C05457=1016.848,96.852,384.023,166.697,54.807,160.034
C05458=1016.842,96.602,384.039,166.694,54.816,160.035
C05459=1016.838,96.353,384.058,166.691,54.825,160.037
C05460=1016.833,96.104,384.074,166.688,54.833,160.038
C05461=1016.828,95.854,384.091,166.685,54.843,160.039
C05462=1016.822,95.605,384.108,166.683,54.852,160.040
C05463=1016.817,95.356,384.125,166.680,54.861,160.041
C05464=1016.813,95.106,384.142,166.677,54.870,160.042
C05465=1016.808,94.857,384.160,166.674,54.880,160.044
C05466=1016.802,94.608,384.177,166.671,54.888,160.045
C05467=1016.797,94.358,384.194,166.669,54.897,160.046
C05468=1016.793,94.109,384.211,166.667,54.906,160.047
C05469=1016.788,93.860,384.228,166.664,54.915,160.048
C05470=1016.783,93.610,384.245,166.661,54.925,160.050
C05471=1016.777,93.361,384.263,166.658,54.933,160.050
C05472=1016.773,93.112,384.280,166.655,54.942,160.052
C05473=1016.768,92.862,384.297,166.652,54.951,160.053
C05474=1016.763,92.613,384.314,166.650,54.961,160.054
C05475=1016.758,92.364,384.331,166.647,54.970,160.055
C05476=1016.753,92.115,384.348,166.645,54.978,160.056
C05477=1016.748,91.865,384.365,166.642,54.987,160.058
C05478=1016.743,91.615,384.382,166.639,54.997,160.059
C05479=1016.738,91.367,384.399,166.637,55.006,160.060
C05480=1016.732,91.085,384.418,166.633,55.015,160.061
C05481=1016.727,90.803,384.438,166.631,55.025,160.063
C05482=1016.722,90.522,384.457,166.627,55.036,160.064
C05483=1016.716,90.240,384.476,166.624,55.046,160.065
C05484=1016.711,89.991,384.493,166.621,55.055,160.066
C05485=1016.706,89.742,384.510,166.619,55.063,160.067
C05486=1016.701,89.492,384.527,166.616,55.073,160.069
C05487=1016.696,89.243,384.544,166.614,55.082,160.070
C05488=1016.692,88.994,384.561,166.611,55.091,160.071
C05489=1016.686,88.744,384.578,166.608,55.100,160.072
C05490=1016.681,88.494,384.594,166.605,55.109,160.073
C05491=1016.676,88.245,384.611,166.602,55.118,160.074
C05492=1016.671,87.996,384.628,166.600,55.127,160.076
C05493=1016.666,87.746,384.645,166.597,55.137,160.077
C05494=1016.661,87.497,384.661,166.594,55.146,160.078
C05495=1016.656,87.247,384.678,166.593,55.155,160.079
C05496=1016.651,86.998,384.695,166.590,55.163,160.080
C05497=1016.646,86.749,384.711,166.587,55.173,160.082
C05498=1016.640,86.500,384.728,166.584,55.182,160.083
C05499=1016.635,86.250,384.744,166.581,55.191,160.084
C05500=1016.631,86.001,384.761,166.579,55.200,160.085
C05501=1016.625,85.751,384.778,166.576,55.210,160.086
C05502=1016.620,85.502,384.795,166.573,55.218,160.087
C05503=1016.616,85.253,384.811,166.570,55.228,160.089
C05504=1016.610,85.003,384.828,166.568,55.237,160.090
C05505=1016.606,84.754,384.844,166.565,55.246,160.091
C05506=1016.601,84.504,384.861,166.562,55.255,160.092
C05507=1016.595,84.255,384.878,166.560,55.263,160.093
C05508=1016.590,84.006,384.894,166.557,55.273,160.095
C05509=1016.585,83.756,384.911,166.555,55.282,160.096
C05510=1016.580,83.507,384.927,166.552,55.291,160.097
C05511=1016.575,83.257,384.943,166.550,55.301,160.098
C05512=1016.570,83.007,384.960,166.546,55.309,160.099
C05513=1016.565,82.759,384.977,166.544,55.318,160.100
C05514=1016.560,82.509,384.994,166.541,55.328,160.102
C05515=1016.556,82.260,385.010,166.539,55.337,160.103
C05516=1016.550,82.010,385.027,166.536,55.345,160.104
C05517=1016.546,81.761,385.043,166.534,55.354,160.105
C05518=1016.540,81.512,385.060,166.531,55.364,160.106
C05519=1016.535,81.262,385.077,166.528,55.372,160.107
C05520=1016.530,81.013,385.092,166.525,55.382,160.109
C05521=1016.525,80.763,385.109,166.523,55.391,160.110
C05522=1016.521,80.514,385.126,166.521,55.400,160.111
C05523=1016.515,80.264,385.143,166.518,55.408,160.112
C05524=1016.511,80.015,385.159,166.515,55.418,160.113
C05525=1016.506,79.766,385.176,166.513,55.427,160.115
C05526=1016.501,79.516,385.192,166.509,55.436,160.116
C05527=1016.496,79.267,385.208,166.507,55.445,160.117
C05528=1016.491,79.018,385.224,166.505,55.454,160.118
C05529=1016.485,78.768,385.241,166.502,55.462,160.119
C05530=1016.481,78.519,385.258,166.499,55.472,160.120
C05531=1016.476,78.269,385.274,166.497,55.481,160.122
C05532=1016.471,78.020,385.290,166.494,55.490,160.123
C05533=1016.466,77.770,385.307,166.492,55.499,160.124
C05534=1016.461,77.521,385.324,166.489,55.507,160.125
C05535=1016.456,77.272,385.341,166.486,55.516,160.126
C05536=1016.452,77.022,385.356,166.484,55.526,160.127
C05537=1016.446,76.773,385.373,166.481,55.534,160.128
C05538=1016.441,76.524,385.389,166.478,55.544,160.130
C05539=1016.436,76.274,385.405,166.477,55.553,160.131
C05540=1016.432,76.025,385.422,166.474,55.562,160.132
C05541=1016.426,75.775,385.438,166.471,55.570,160.133
C05542=1016.422,75.526,385.454,166.468,55.580,160.134
C05543=1016.416,75.276,385.470,166.466,55.589,160.136
C05544=1016.411,74.995,385.488,166.463,55.600,160.137
C05545=1016.404,74.713,385.506,166.460,55.610,160.138
C05546=1016.399,74.432,385.525,166.457,55.619,160.139
C05547=1016.393,74.151,385.543,166.454,55.630,160.141
C05548=1016.388,73.901,385.559,166.451,55.639,160.142
C05549=1016.383,73.652,385.575,166.449,55.649,160.143
C05550=1016.378,73.402,385.591,166.445,55.657,160.144
C05551=1016.373,73.153,385.607,166.444,55.666,160.146
C05552=1016.368,72.904,385.623,166.441,55.675,160.147
C05553=1016.363,72.654,385.639,166.438,55.684,160.148
C05554=1016.358,72.405,385.655,166.436,55.693,160.149
C05555=1016.353,72.155,385.671,166.433,55.703,160.150
C05556=1016.348,71.906,385.688,166.430,55.711,160.151
C05557=1016.343,71.656,385.703,166.428,55.721,160.152
C05558=1016.338,71.407,385.720,166.426,55.730,160.154
C05559=1016.333,71.158,385.735,166.423,55.738,160.155
C05560=1016.328,70.908,385.752,166.420,55.748,160.156
C05561=1016.323,70.659,385.768,166.418,55.757,160.157
C05562=1016.318,70.409,385.784,166.415,55.766,160.158
C05563=1016.313,70.160,385.800,166.412,55.775,160.159
C05564=1016.308,69.911,385.815,166.411,55.784,160.161
C05565=1016.303,69.661,385.832,166.408,55.793,160.162
C05566=1016.298,69.412,385.847,166.405,55.802,160.163
C05567=1016.293,69.162,385.864,166.403,55.811,160.164
C05568=1016.288,68.912,385.880,166.399,55.820,160.165
C05569=1016.283,68.664,385.896,166.397,55.829,160.167
C05570=1016.278,68.414,385.912,166.395,55.837,160.168
C05571=1016.273,68.164,385.927,166.392,55.847,160.169
C05572=1016.269,67.915,385.943,166.390,55.856,160.170
C05573=1016.263,67.665,385.959,166.387,55.865,160.171
C05574=1016.259,67.416,385.975,166.384,55.874,160.172
C05575=1016.253,67.167,385.991,166.382,55.884,160.174
C05576=1016.248,66.917,386.006,166.380,55.892,160.175
C05577=1016.243,66.668,386.022,166.377,55.901,160.176
C05578=1016.237,66.418,386.038,166.375,55.911,160.177
C05579=1016.233,66.169,386.054,166.372,55.919,160.178
C05580=1016.228,65.919,386.069,166.369,55.929,160.179
C05581=1016.222,65.670,386.085,166.367,55.938,160.181
C05582=1016.218,65.420,386.101,166.364,55.947,160.182
C05583=1016.213,65.171,386.116,166.362,55.956,160.183
C05584=1016.208,64.921,386.132,166.359,55.964,160.184
C05585=1016.202,64.672,386.148,166.357,55.974,160.185
C05586=1016.197,64.423,386.163,166.354,55.983,160.187
C05587=1016.192,64.173,386.180,166.351,55.992,160.188
C05588=1016.187,63.923,386.195,166.349,56.001,160.189
C05589=1016.182,63.674,386.210,166.346,56.011,160.190
C05590=1016.178,63.425,386.226,166.344,56.019,160.191
C05591=1016.172,63.175,386.242,166.342,56.028,160.192
C05592=1016.167,62.926,386.257,166.339,56.037,160.193
C05593=1016.163,62.676,386.273,166.336,56.046,160.195
C05594=1016.157,62.426,386.288,166.334,56.056,160.196
C05595=1016.152,62.177,386.304,166.331,56.064,160.197
C05596=1016.147,61.928,386.319,166.328,56.074,160.198
C05597=1016.141,61.678,386.334,166.326,56.083,160.199
C05598=1016.136,61.429,386.349,166.323,56.093,160.201
C05599=1016.131,61.179,386.365,166.320,56.101,160.202
C05600=1016.126,60.930,386.380,166.318,56.111,160.203
C05601=1016.121,60.680,386.395,166.316,56.120,160.204
C05602=1016.116,60.431,386.411,166.314,56.129,160.206
C05603=1016.111,60.182,386.426,166.311,56.138,160.206
C05604=1016.105,59.932,386.441,166.308,56.147,160.208
C05605=1016.100,59.682,386.456,166.306,56.157,160.209
C05606=1016.096,59.433,386.472,166.303,56.166,160.210
C05607=1016.090,59.184,386.487,166.300,56.175,160.211
C05608=1016.084,58.903,386.504,166.298,56.185,160.213
C05609=1016.079,58.621,386.521,166.295,56.196,160.214
C05610=1016.073,58.340,386.539,166.293,56.206,160.215
C05611=1016.067,58.058,386.556,166.289,56.216,160.217
C05612=1016.062,57.808,386.571,166.287,56.225,160.218
C05613=1016.057,57.559,386.587,166.284,56.235,160.219
C05614=1016.052,57.310,386.602,166.281,56.243,160.220
C05615=1016.047,57.060,386.617,166.279,56.253,160.221
C05616=1016.042,56.811,386.632,166.276,56.262,160.223
C05617=1016.036,56.561,386.648,166.273,56.271,160.224
C05618=1016.031,56.312,386.663,166.272,56.280,160.225
C05619=1016.026,56.063,386.678,166.269,56.289,160.226
C05620=1016.021,55.813,386.693,166.267,56.298,160.227
C05621=1016.016,55.563,386.708,166.264,56.307,160.228
C05622=1016.010,55.314,386.723,166.261,56.316,160.229
C05623=1016.005,55.064,386.738,166.259,56.326,160.231
C05624=1016.000,54.815,386.754,166.256,56.334,160.232
C05625=1015.995,54.566,386.769,166.253,56.344,160.233
C05626=1015.990,54.316,386.784,166.252,56.352,160.234
C05627=1015.985,54.067,386.799,166.249,56.361,160.235
C05628=1015.980,53.817,386.814,166.246,56.370,160.236
C05629=1015.975,53.567,386.829,166.244,56.380,160.238
C05630=1015.970,53.318,386.844,166.241,56.388,160.239
C05631=1015.965,53.069,386.859,166.238,56.398,160.240
C05632=1015.960,52.820,386.875,166.237,56.406,160.241
C05633=1015.955,52.570,386.890,166.234,56.416,160.242
C05634=1015.950,52.320,386.904,166.231,56.424,160.243
C05635=1015.945,52.070,386.920,166.229,56.434,160.245
C05636=1015.940,51.821,386.936,166.226,56.442,160.246
C05637=1015.935,51.572,386.951,166.225,56.452,160.247
C05638=1015.930,51.322,386.966,166.222,56.460,160.248
C05639=1015.925,51.072,386.980,166.219,56.470,160.249
C05640=1015.920,50.823,386.996,166.216,56.478,160.250
C05641=1015.915,50.574,387.011,166.214,56.488,160.252
C05642=1015.910,50.325,387.026,166.212,56.496,160.253
C05643=1015.905,50.074,387.041,166.209,56.505,160.254
C05644=1015.900,49.825,387.056,166.207,56.514,160.255
C05645=1015.895,49.575,387.071,166.204,56.523,160.256
C05646=1015.889,49.326,387.086,166.201,56.533,160.257
C05647=1015.885,49.076,387.101,166.200,56.541,160.258
C05648=1015.880,48.827,387.116,166.197,56.550,160.259
C05649=1015.875,48.578,387.131,166.194,56.559,160.261
C05650=1015.870,48.329,387.146,166.191,56.568,160.262
C05651=1015.865,48.079,387.161,166.189,56.576,160.263
C05652=1015.860,47.829,387.176,166.187,56.586,160.264
C05653=1015.855,47.580,387.191,166.184,56.594,160.265
C05654=1015.850,47.331,387.206,166.181,56.603,160.266
C05655=1015.845,47.081,387.221,166.180,56.612,160.268
C05656=1015.839,46.831,387.236,166.177,56.621,160.268
C05657=1015.834,46.582,387.251,166.174,56.630,160.269
C05658=1015.830,46.332,387.266,166.171,56.639,160.270
C05659=1015.825,46.083,387.281,166.170,56.648,160.272
C05660=1015.819,45.833,387.296,166.167,56.656,160.273
C05661=1015.815,45.583,387.311,166.164,56.665,160.274
C05662=1015.810,45.334,387.326,166.163,56.674,160.275
C05663=1015.805,45.085,387.341,166.160,56.683,160.276
C05664=1015.800,44.835,387.355,166.157,56.692,160.277
C05665=1015.795,44.586,387.371,166.154,56.701,160.278
C05666=1015.790,44.336,387.386,166.152,56.709,160.280
C05667=1015.785,44.087,387.400,166.150,56.718,160.281
C05668=1015.780,43.837,387.415,166.147,56.727,160.282
C05669=1015.775,43.587,387.430,166.145,56.736,160.283
C05670=1015.770,43.338,387.445,166.143,56.744,160.284
C05671=1015.765,43.089,387.460,166.140,56.753,160.285
C05672=1015.760,42.831,387.476,166.138,56.762,160.286
C05673=1015.755,42.574,387.491,166.135,56.771,160.287
C05674=1015.751,42.315,387.506,166.133,56.780,160.289
C05675=1015.745,42.058,387.521,166.130,56.789,160.290
C05676=1015.740,41.809,387.536,166.127,56.798,160.291
C05677=1015.735,41.559,387.551,166.125,56.807,160.292
C05678=1015.730,41.310,387.565,166.122,56.816,160.293
C05679=1015.725,41.060,387.580,166.120,56.825,160.294
C05680=1015.720,40.810,387.594,166.118,56.834,160.295
C05681=1015.715,40.561,387.610,166.115,56.843,160.296
C05682=1015.710,40.311,387.623,166.112,56.852,160.297
C05683=1015.705,40.062,387.639,166.111,56.861,160.299
C05684=1015.701,39.813,387.653,166.108,56.870,160.300
C05685=1015.695,39.563,387.667,166.105,56.878,160.301
C05686=1015.690,39.314,387.682,166.103,56.887,160.302
C05687=1015.685,39.064,387.696,166.101,56.896,160.303
C05688=1015.680,38.815,387.711,166.099,56.905,160.304
C05689=1015.675,38.565,387.725,166.096,56.914,160.305
C05690=1015.670,38.315,387.740,166.093,56.923,160.306
C05691=1015.665,38.066,387.755,166.092,56.932,160.308
C05692=1015.660,37.816,387.769,166.089,56.941,160.309
C05693=1015.655,37.567,387.783,166.086,56.949,160.310
C05694=1015.650,37.317,387.798,166.083,56.958,160.311
C05695=1015.645,37.068,387.813,166.081,56.967,160.312
C05696=1015.639,36.818,387.827,166.079,56.976,160.313
C05697=1015.635,36.568,387.841,166.076,56.985,160.314
C05698=1015.630,36.319,387.856,166.074,56.993,160.316
C05699=1015.625,36.070,387.870,166.072,57.002,160.317
C05700=1015.620,35.820,387.884,166.069,57.012,160.318
C05701=1015.615,35.571,387.898,166.067,57.020,160.319
C05702=1015.610,35.321,387.913,166.064,57.029,160.320
C05703=1015.604,35.072,387.927,166.061,57.038,160.321
C05704=1015.599,34.822,387.942,166.060,57.047,160.322
C05705=1015.594,34.572,387.956,166.057,57.056,160.323
C05706=1015.589,34.322,387.970,166.054,57.065,160.324
C05707=1015.584,34.073,387.983,166.051,57.074,160.325
C05708=1015.580,33.824,387.998,166.049,57.083,160.327
C05709=1015.574,33.574,388.012,166.047,57.092,160.328
C05710=1015.569,33.325,388.027,166.044,57.100,160.329
C05711=1015.564,33.075,388.041,166.042,57.109,160.330
C05712=1015.558,32.826,388.055,166.039,57.119,160.331
C05713=1015.553,32.576,388.069,166.038,57.127,160.332
C05714=1015.548,32.327,388.083,166.035,57.136,160.333
C05715=1015.544,32.077,388.097,166.032,57.145,160.334
C05716=1015.538,31.827,388.111,166.029,57.154,160.335
C05717=1015.533,31.577,388.125,166.028,57.163,160.337
C05718=1015.528,31.328,388.139,166.025,57.172,160.338
C05719=1015.523,31.078,388.154,166.023,57.181,160.339
C05720=1015.518,30.829,388.167,166.020,57.189,160.340
C05721=1015.513,30.580,388.182,166.018,57.198,160.341
C05722=1015.508,30.330,388.196,166.015,57.207,160.342
C05723=1015.503,30.080,388.211,166.012,57.215,160.343
C05724=1015.498,29.807,388.226,166.010,57.225,160.345
C05725=1015.492,29.534,388.241,166.007,57.235,160.346
C05726=1015.487,29.260,388.256,166.005,57.245,160.347
C05727=1015.481,28.987,388.271,166.003,57.254,160.348
C05728=1015.476,28.737,388.286,166.000,57.263,160.349
C05729=1015.471,28.488,388.299,165.997,57.272,160.350
C05730=1015.467,28.238,388.314,165.995,57.280,160.352
C05731=1015.461,27.989,388.328,165.993,57.289,160.353
C05732=1015.456,27.739,388.342,165.990,57.298,160.354
C05733=1015.451,27.490,388.356,165.988,57.306,160.355
C05734=1015.446,27.240,388.370,165.985,57.315,160.356
C05735=1015.441,26.990,388.384,165.983,57.324,160.357
C05736=1015.436,26.710,388.400,165.980,57.334,160.358
C05737=1015.429,26.428,388.415,165.977,57.344,160.359
C05738=1015.423,26.147,388.431,165.975,57.355,160.361
C05739=1015.418,25.866,388.446,165.972,57.364,160.362
C05740=1015.413,25.616,388.460,165.970,57.373,160.363
C05741=1015.408,25.366,388.475,165.967,57.382,160.364
C05742=1015.403,25.116,388.488,165.965,57.390,160.365
C05743=1015.398,24.867,388.501,165.962,57.399,160.366
C05744=1015.392,24.618,388.515,165.960,57.408,160.367
C05745=1015.388,24.368,388.530,165.957,57.417,160.368
C05746=1015.383,24.119,388.543,165.955,57.425,160.369
C05747=1015.378,23.869,388.556,165.953,57.434,160.370
C05748=1015.372,23.619,388.570,165.950,57.443,160.371
C05749=1015.367,23.370,388.584,165.947,57.452,160.373
C05750=1015.363,23.120,388.598,165.945,57.460,160.374
C05751=1015.357,22.871,388.612,165.943,57.469,160.375
C05752=1015.352,22.621,388.625,165.940,57.478,160.376
C05753=1015.347,22.372,388.639,165.938,57.487,160.377
C05754=1015.342,22.122,388.652,165.935,57.495,160.378
C05755=1015.337,21.872,388.666,165.933,57.504,160.379
C05756=1015.332,21.623,388.680,165.930,57.513,160.380
C05757=1015.327,21.373,388.693,165.928,57.522,160.381
C05758=1015.321,21.124,388.707,165.926,57.531,160.382
C05759=1015.317,20.874,388.720,165.923,57.539,160.383
C05760=1015.312,20.624,388.735,165.921,57.548,160.385
C05761=1015.307,20.375,388.748,165.919,57.557,160.386
C05762=1015.302,20.125,388.761,165.916,57.566,160.387
C05763=1015.297,19.876,388.775,165.914,57.574,160.388
C05764=1015.291,19.626,388.789,165.912,57.583,160.389
C05765=1015.287,19.377,388.803,165.908,57.591,160.390
C05766=1015.282,19.127,388.816,165.907,57.600,160.391
C05767=1015.277,18.878,388.830,165.904,57.609,160.392
C05768=1015.272,18.628,388.843,165.901,57.617,160.393
C05769=1015.266,18.378,388.857,165.900,57.626,160.394
C05770=1015.261,18.129,388.870,165.897,57.635,160.395
C05771=1015.256,17.879,388.883,165.894,57.644,160.396
C05772=1015.251,17.630,388.897,165.893,57.652,160.397
C05773=1015.246,17.380,388.910,165.890,57.661,160.398
C05774=1015.241,17.130,388.924,165.887,57.670,160.399
C05775=1015.236,16.881,388.937,165.884,57.679,160.400
C05776=1015.231,16.631,388.951,165.882,57.687,160.401
C05777=1015.227,16.381,388.964,165.880,57.696,160.402
C05778=1015.221,16.132,388.978,165.877,57.704,160.403
C05779=1015.216,15.882,388.992,165.875,57.713,160.405
C05780=1015.211,15.633,389.004,165.873,57.722,160.406
C05781=1015.206,15.383,389.018,165.870,57.731,160.407
C05782=1015.201,15.134,389.031,165.868,57.739,160.408
C05783=1015.196,14.884,389.045,165.865,57.747,160.409
C05784=1015.191,14.635,389.058,165.863,57.756,160.410
C05785=1015.186,14.385,389.072,165.861,57.765,160.411
C05786=1015.181,14.135,389.085,165.858,57.774,160.412
C05787=1015.176,13.886,389.098,165.856,57.781,160.413
C05788=1015.170,13.636,389.111,165.853,57.790,160.414
C05789=1015.166,13.386,389.124,165.850,57.799,160.415
C05790=1015.160,13.137,389.138,165.849,57.808,160.416
C05791=1015.156,12.887,389.151,165.846,57.817,160.417
C05792=1015.151,12.637,389.164,165.844,57.826,160.418
C05793=1015.145,12.388,389.178,165.841,57.833,160.419
C05794=1015.140,12.138,389.190,165.839,57.842,160.420
C05795=1015.135,11.888,389.203,165.836,57.851,160.421
C05796=1015.130,11.639,389.217,165.833,57.860,160.422
C05797=1015.125,11.389,389.230,165.832,57.869,160.424
C05798=1015.119,11.140,389.242,165.829,57.878,160.425
C05799=1015.114,10.890,389.255,165.827,57.887,160.426
C05800=1015.108,10.610,389.270,165.825,57.896,160.427
C05801=1015.103,10.331,389.285,165.821,57.906,160.428
C05802=1015.097,10.051,389.298,165.819,57.915,160.429
C05803=1015.091,9.771,389.313,165.816,57.925,160.430
C05804=1015.086,9.521,389.327,165.813,57.934,160.431
C05805=1015.082,9.272,389.339,165.811,57.942,160.432
C05806=1015.076,9.022,389.353,165.808,57.951,160.433
C05807=1015.071,8.773,389.365,165.806,57.960,160.434
C05808=1015.066,8.523,389.379,165.804,57.968,160.436
C05809=1015.061,8.273,389.391,165.801,57.977,160.436
C05810=1015.056,8.024,389.404,165.798,57.986,160.437
C05811=1015.050,7.774,389.417,165.797,57.994,160.439
C05812=1015.046,7.525,389.430,165.794,58.003,160.440
C05813=1015.041,7.275,389.443,165.791,58.011,160.440
C05814=1015.035,7.026,389.456,165.789,58.020,160.442
C05815=1015.030,6.775,389.469,165.787,58.029,160.443
C05816=1015.026,6.526,389.481,165.784,58.037,160.444
C05817=1015.021,6.276,389.494,165.782,58.046,160.445
C05818=1015.015,6.027,389.508,165.779,58.054,160.446
C05819=1015.010,5.778,389.520,165.777,58.062,160.447
C05820=1015.005,5.527,389.533,165.774,58.071,160.448
C05821=1015.001,5.278,389.546,165.773,58.080,160.449
C05822=1014.995,5.028,389.559,165.770,58.088,160.450
C05823=1014.990,4.779,389.572,165.767,58.097,160.451
C05824=1014.986,4.529,389.584,165.765,58.105,160.452
C05825=1014.980,4.279,389.598,165.762,58.114,160.453
C05826=1014.975,4.030,389.610,165.761,58.122,160.454
C05827=1014.970,3.781,389.623,165.758,58.130,160.455
C05828=1014.965,3.531,389.636,165.755,58.139,160.456
C05829=1014.960,3.281,389.649,165.753,58.147,160.457
C05830=1014.955,3.031,389.662,165.750,58.156,160.458
C05831=1014.950,2.782,389.674,165.748,58.164,160.459
C05832=1014.945,2.532,389.687,165.746,58.173,160.460
C05833=1014.940,2.282,389.700,165.743,58.181,160.461
C05834=1014.935,2.033,389.713,165.741,58.190,160.462
C05835=1014.930,1.783,389.725,165.739,58.198,160.463
C05836=1014.925,1.533,389.739,165.736,58.206,160.464
C05837=1014.920,1.284,389.751,165.734,58.214,160.465
C05838=1014.915,1.035,389.763,165.731,58.223,160.465
C05839=1014.910,0.784,389.777,165.729,58.231,160.467
C05840=1014.906,0.535,389.789,165.726,58.239,160.467
C05841=1014.900,0.286,389.802,165.725,58.248,160.469
C05842=1014.895,0.035,389.815,165.722,58.256,160.469
C05843=1014.890,-0.214,389.828,165.719,58.264,160.470
C05844=1014.886,-0.464,389.840,165.717,58.273,160.471
C05845=1014.880,-0.713,389.853,165.715,58.281,160.472
C05846=1014.875,-0.963,389.866,165.712,58.290,160.473
C05847=1014.871,-1.212,389.878,165.710,58.298,160.474
C05848=1014.866,-1.462,389.891,165.707,58.306,160.475
C05849=1014.860,-1.712,389.904,165.705,58.314,160.476
C05850=1014.856,-1.961,389.917,165.702,58.323,160.477
C05851=1014.851,-2.211,389.929,165.700,58.330,160.478
C05852=1014.845,-2.461,389.942,165.697,58.339,160.479
C05853=1014.841,-2.710,389.955,165.695,58.347,160.480
C05854=1014.836,-2.960,389.967,165.693,58.355,160.481
C05855=1014.832,-3.209,389.980,165.690,58.363,160.482
C05856=1014.826,-3.459,389.993,165.688,58.371,160.483
C05857=1014.821,-3.708,390.006,165.686,58.380,160.484
C05858=1014.817,-3.958,390.018,165.683,58.388,160.485
C05859=1014.812,-4.207,390.031,165.680,58.396,160.485
C05860=1014.806,-4.458,390.043,165.678,58.404,160.486
C05861=1014.802,-4.707,390.056,165.677,58.413,160.487
C05862=1014.797,-4.957,390.068,165.674,58.421,160.488
C05863=1014.792,-5.206,390.081,165.670,58.429,160.489
C05864=1014.786,-5.484,390.094,165.669,58.439,160.490
C05865=1014.781,-5.762,390.107,165.666,58.448,160.491
C05866=1014.775,-6.039,390.121,165.663,58.457,160.492
C05867=1014.769,-6.317,390.135,165.660,58.466,160.493
C05868=1014.764,-6.566,390.146,165.658,58.475,160.495
C05869=1014.759,-6.817,390.160,165.655,58.483,160.495
C05870=1014.754,-7.066,390.172,165.653,58.491,160.496
C05871=1014.749,-7.316,390.183,165.651,58.500,160.497
C05872=1014.744,-7.565,390.196,165.649,58.508,160.498
C05873=1014.739,-7.815,390.207,165.646,58.516,160.499
C05874=1014.733,-8.065,390.220,165.644,58.525,160.500
C05875=1014.729,-8.314,390.233,165.641,58.533,160.501
C05876=1014.724,-8.564,390.244,165.639,58.541,160.502
C05877=1014.718,-8.813,390.256,165.636,58.549,160.503
C05878=1014.714,-9.063,390.269,165.634,58.558,160.504
C05879=1014.709,-9.313,390.281,165.631,58.566,160.505
C05880=1014.704,-9.563,390.294,165.629,58.574,160.506
C05881=1014.699,-9.813,390.305,165.626,58.582,160.506
C05882=1014.693,-10.062,390.318,165.625,58.591,160.508
C05883=1014.689,-10.312,390.330,165.621,58.599,160.508
C05884=1014.684,-10.561,390.342,165.619,58.607,160.509
C05885=1014.678,-10.810,390.354,165.616,58.615,160.510
C05886=1014.674,-11.060,390.366,165.614,58.623,160.511
C05887=1014.668,-11.310,390.379,165.612,58.631,160.512
C05888=1014.663,-11.560,390.390,165.610,58.640,160.513
C05889=1014.659,-11.810,390.403,165.608,58.648,160.514
C05890=1014.654,-12.059,390.414,165.605,58.656,160.515
C05891=1014.648,-12.309,390.427,165.602,58.664,160.516
C05892=1014.644,-12.559,390.439,165.600,58.672,160.517
C05893=1014.639,-12.808,390.451,165.597,58.680,160.518
C05894=1014.634,-13.058,390.462,165.595,58.688,160.518
C05895=1014.629,-13.307,390.475,165.592,58.696,160.519
C05896=1014.624,-13.557,390.487,165.590,58.704,160.520
C05897=1014.619,-13.806,390.499,165.588,58.712,160.521
C05898=1014.614,-14.057,390.511,165.585,58.720,160.522
C05899=1014.609,-14.306,390.523,165.583,58.728,160.523
C05900=1014.604,-14.556,390.535,165.581,58.736,160.524
C05901=1014.599,-14.805,390.548,165.578,58.744,160.525
C05902=1014.594,-15.055,390.559,165.576,58.752,160.526
C05903=1014.589,-15.305,390.571,165.574,58.760,160.526
C05904=1014.585,-15.554,390.583,165.571,58.768,160.527
C05905=1014.580,-15.804,390.595,165.569,58.776,160.528
C05906=1014.575,-16.054,390.608,165.567,58.784,160.529
C05907=1014.570,-16.304,390.619,165.564,58.792,160.530
C05908=1014.565,-16.553,390.630,165.562,58.800,160.531
C05909=1014.560,-16.803,390.642,165.559,58.809,160.532
C05910=1014.555,-17.052,390.654,165.557,58.817,160.533
C05911=1014.550,-17.302,390.666,165.553,58.825,160.533
C05912=1014.545,-17.552,390.677,165.551,58.833,160.534
C05913=1014.540,-17.802,390.689,165.549,58.841,160.535
C05914=1014.534,-18.051,390.701,165.546,58.849,160.536
C05915=1014.529,-18.301,390.712,165.544,58.857,160.537
C05916=1014.524,-18.551,390.724,165.541,58.865,160.538
C05917=1014.519,-18.800,390.735,165.539,58.873,160.539
C05918=1014.515,-19.050,390.748,165.537,58.881,160.540
C05919=1014.510,-19.300,390.759,165.534,58.889,160.540
C05920=1014.505,-19.549,390.771,165.532,58.897,160.541
C05921=1014.500,-19.799,390.782,165.530,58.905,160.542
C05922=1014.495,-20.049,390.794,165.527,58.913,160.543
C05923=1014.489,-20.298,390.806,165.525,58.921,160.544
C05924=1014.484,-20.548,390.818,165.523,58.929,160.545
C05925=1014.479,-20.798,390.829,165.520,58.937,160.546
C05926=1014.474,-21.048,390.840,165.518,58.945,160.547
C05927=1014.469,-21.297,390.852,165.516,58.953,160.548
C05928=1014.464,-21.573,390.865,165.513,58.962,160.548
C05929=1014.458,-21.849,390.878,165.511,58.971,160.550
C05930=1014.453,-22.125,390.891,165.508,58.979,160.550
C05931=1014.448,-22.401,390.903,165.505,58.988,160.551
C05932=1014.443,-22.651,390.915,165.502,58.996,160.552
C05933=1014.438,-22.900,390.927,165.499,59.004,160.553
C05934=1014.433,-23.150,390.938,165.498,59.011,160.554
C05935=1014.428,-23.399,390.950,165.496,59.019,160.555
C05936=1014.423,-23.649,390.961,165.492,59.028,160.555
C05937=1014.418,-23.899,390.973,165.490,59.035,160.556
C05938=1014.413,-24.148,390.984,165.488,59.043,160.557
C05939=1014.408,-24.398,390.995,165.486,59.051,160.558
C05940=1014.403,-24.648,391.007,165.483,59.059,160.559
C05941=1014.398,-24.897,391.018,165.480,59.066,160.559
C05942=1014.393,-25.147,391.030,165.478,59.074,160.560
C05943=1014.388,-25.397,391.041,165.476,59.082,160.561
C05944=1014.383,-25.647,391.053,165.473,59.090,160.562
C05945=1014.378,-25.897,391.064,165.471,59.097,160.563
C05946=1014.374,-26.146,391.075,165.469,59.105,160.564
C05947=1014.369,-26.395,391.088,165.466,59.113,160.564
C05948=1014.364,-26.645,391.100,165.464,59.120,160.565
C05949=1014.359,-26.895,391.111,165.462,59.128,160.566
C05950=1014.354,-27.145,391.122,165.459,59.136,160.567
C05951=1014.349,-27.394,391.134,165.456,59.143,160.567
C05952=1014.345,-27.644,391.145,165.454,59.151,160.568
C05953=1014.340,-27.894,391.156,165.452,59.159,160.569
C05954=1014.335,-28.144,391.167,165.449,59.166,160.570
C05955=1014.329,-28.393,391.178,165.446,59.175,160.571
C05956=1014.324,-28.643,391.190,165.445,59.182,160.572
C05957=1014.319,-28.893,391.201,165.442,59.190,160.572
C05958=1014.315,-29.142,391.212,165.440,59.198,160.573
C05959=1014.310,-29.392,391.222,165.437,59.206,160.574
C05960=1014.305,-29.642,391.234,165.434,59.213,160.575
C05961=1014.300,-29.892,391.245,165.432,59.221,160.576
C05962=1014.295,-30.141,391.257,165.431,59.229,160.577
C05963=1014.290,-30.391,391.268,165.427,59.237,160.577
C05964=1014.285,-30.641,391.278,165.425,59.244,160.578
C05965=1014.280,-30.890,391.290,165.422,59.252,160.579
C05966=1014.275,-31.140,391.301,165.420,59.260,160.580
C05967=1014.270,-31.389,391.312,165.417,59.268,160.580
C05968=1014.265,-31.640,391.322,165.415,59.275,160.581
C05969=1014.260,-31.889,391.334,165.413,59.283,160.582
C05970=1014.255,-32.139,391.345,165.410,59.290,160.583
C05971=1014.251,-32.388,391.356,165.408,59.298,160.584
C05972=1014.245,-32.638,391.366,165.406,59.305,160.584
C05973=1014.240,-32.888,391.378,165.403,59.314,160.585
C05974=1014.236,-33.137,391.389,165.400,59.321,160.586
C05975=1014.231,-33.388,391.400,165.398,59.329,160.587
C05976=1014.225,-33.637,391.411,165.396,59.336,160.587
C05977=1014.220,-33.887,391.422,165.393,59.343,160.588
C05978=1014.216,-34.136,391.433,165.391,59.351,160.589
C05979=1014.211,-34.386,391.444,165.389,59.358,160.590
C05980=1014.205,-34.636,391.455,165.387,59.366,160.591
C05981=1014.201,-34.885,391.466,165.383,59.374,160.591
C05982=1014.196,-35.135,391.477,165.381,59.381,160.592
C05983=1014.191,-35.385,391.488,165.379,59.389,160.593
C05984=1014.186,-35.634,391.499,165.376,59.396,160.593
C05985=1014.182,-35.884,391.510,165.374,59.404,160.594
C05986=1014.177,-36.134,391.521,165.372,59.411,160.595
C05987=1014.172,-36.384,391.531,165.369,59.419,160.596
C05988=1014.167,-36.633,391.542,165.367,59.426,160.596
C05989=1014.162,-36.883,391.554,165.365,59.434,160.597
C05990=1014.158,-37.133,391.564,165.362,59.441,160.598
C05991=1014.153,-37.383,391.576,165.360,59.448,160.599
C05992=1014.147,-37.657,391.588,165.357,59.457,160.599
C05993=1014.142,-37.932,391.600,165.355,59.465,160.600
C05994=1014.137,-38.208,391.612,165.352,59.473,160.601
C05995=1014.131,-38.482,391.623,165.348,59.481,160.601
C05996=1014.126,-38.731,391.634,165.347,59.488,160.603
C05997=1014.121,-38.982,391.645,165.345,59.495,160.603
C05998=1014.116,-39.231,391.656,165.342,59.503,160.604
C05999=1014.112,-39.481,391.666,165.340,59.510,160.605
C06000=1014.107,-39.731,391.678,165.337,59.517,160.605
C06001=1014.103,-39.980,391.688,165.334,59.525,160.606
C06002=1014.097,-40.230,391.699,165.332,59.533,160.607
C06003=1014.091,-40.480,391.709,165.329,59.540,160.607
C06004=1014.087,-40.730,391.719,165.327,59.547,160.608
C06005=1014.081,-40.979,391.730,165.325,59.555,160.609
C06006=1014.077,-41.229,391.741,165.322,59.562,160.610
C06007=1014.072,-41.479,391.751,165.320,59.569,160.610
C06008=1014.068,-41.728,391.762,165.317,59.577,160.611
C06009=1014.062,-41.978,391.772,165.315,59.585,160.612
C06010=1014.058,-42.227,391.783,165.313,59.592,160.613
C06011=1014.052,-42.477,391.793,165.310,59.599,160.613
C06012=1014.048,-42.728,391.804,165.308,59.606,160.614
C06013=1014.042,-42.977,391.815,165.305,59.613,160.615
C06014=1014.038,-43.227,391.825,165.303,59.621,160.615
C06015=1014.033,-43.476,391.835,165.300,59.628,160.616
C06016=1014.028,-43.727,391.846,165.298,59.636,160.617
C06017=1014.023,-43.976,391.857,165.296,59.643,160.618
C06018=1014.018,-44.226,391.867,165.293,59.650,160.618
C06019=1014.014,-44.475,391.877,165.291,59.658,160.619
C06020=1014.008,-44.725,391.888,165.288,59.665,160.619
C06021=1014.004,-44.975,391.898,165.286,59.672,160.620
C06022=1013.998,-45.225,391.909,165.283,59.679,160.621
C06023=1013.994,-45.474,391.919,165.282,59.686,160.622
C06024=1013.988,-45.724,391.930,165.279,59.693,160.622
C06025=1013.984,-45.974,391.940,165.277,59.700,160.623
C06026=1013.979,-46.224,391.950,165.274,59.708,160.624
C06027=1013.975,-46.473,391.961,165.272,59.715,160.624
C06028=1013.970,-46.722,391.971,165.269,59.722,160.625
C06029=1013.965,-46.973,391.982,165.267,59.729,160.626
C06030=1013.960,-47.222,391.992,165.263,59.736,160.626
C06031=1013.956,-47.473,392.003,165.262,59.743,160.627
C06032=1013.951,-47.722,392.012,165.259,59.750,160.627
C06033=1013.945,-47.971,392.023,165.257,59.757,160.628
C06034=1013.941,-48.221,392.034,165.254,59.764,160.629
C06035=1013.935,-48.471,392.044,165.252,59.772,160.629
C06036=1013.931,-48.721,392.054,165.249,59.779,160.630
C06037=1013.926,-48.970,392.064,165.247,59.785,160.631
C06038=1013.921,-49.220,392.075,165.245,59.792,160.631
C06039=1013.917,-49.470,392.085,165.242,59.799,160.632
C06040=1013.912,-49.720,392.096,165.240,59.807,160.633
C06041=1013.907,-49.969,392.106,165.237,59.814,160.633
C06042=1013.903,-50.219,392.116,165.235,59.820,160.634
C06043=1013.898,-50.469,392.126,165.233,59.827,160.634
C06044=1013.893,-50.719,392.137,165.230,59.834,160.635
C06045=1013.888,-50.969,392.147,165.227,59.841,160.635
C06046=1013.884,-51.219,392.157,165.226,59.848,160.636
C06047=1013.879,-51.469,392.167,165.223,59.855,160.637
C06048=1013.874,-51.718,392.177,165.221,59.862,160.638
C06049=1013.869,-51.968,392.187,165.218,59.869,160.638
C06050=1013.863,-52.218,392.197,165.216,59.877,160.639
C06051=1013.859,-52.467,392.207,165.213,59.884,160.639
C06052=1013.854,-52.717,392.217,165.211,59.891,160.640
C06053=1013.849,-52.967,392.226,165.208,59.898,160.640
C06054=1013.844,-53.217,392.236,165.206,59.904,160.641
C06055=1013.839,-53.466,392.246,165.204,59.912,160.642
C06056=1013.833,-53.741,392.257,165.201,59.920,160.643
C06057=1013.828,-54.016,392.268,165.198,59.927,160.643
C06058=1013.823,-54.291,392.279,165.195,59.935,160.644
C06059=1013.817,-54.567,392.289,165.193,59.943,160.645
C06060=1013.812,-54.817,392.299,165.190,59.950,160.645
C06061=1013.807,-55.066,392.309,165.187,59.957,160.646
C06062=1013.802,-55.315,392.319,165.186,59.964,160.647
C06063=1013.797,-55.565,392.328,165.183,59.971,160.647
C06064=1013.792,-55.816,392.338,165.180,59.978,160.648
C06065=1013.787,-56.065,392.348,165.178,59.985,160.648
C06066=1013.783,-56.314,392.357,165.175,59.992,160.649
C06067=1013.777,-56.565,392.368,165.173,59.998,160.649
C06068=1013.773,-56.815,392.377,165.171,60.005,160.650
C06069=1013.768,-57.064,392.386,165.168,60.013,160.651
C06070=1013.764,-57.314,392.397,165.166,60.019,160.651
C06071=1013.758,-57.564,392.407,165.164,60.026,160.652
C06072=1013.754,-57.814,392.416,165.161,60.033,160.653
C06073=1013.749,-58.063,392.426,165.158,60.040,160.653
C06074=1013.744,-58.313,392.436,165.157,60.047,160.654
C06075=1013.740,-58.563,392.445,165.154,60.053,160.654
C06076=1013.734,-58.813,392.455,165.151,60.060,160.655
C06077=1013.729,-59.062,392.465,165.149,60.066,160.655
C06078=1013.724,-59.312,392.475,165.147,60.074,160.656
C06079=1013.720,-59.562,392.484,165.144,60.080,160.656
C06080=1013.714,-59.812,392.494,165.142,60.087,160.657
C06081=1013.710,-60.061,392.504,165.139,60.094,160.658
C06082=1013.705,-60.311,392.513,165.137,60.101,160.658
C06083=1013.700,-60.561,392.522,165.135,60.107,160.659
C06084=1013.695,-60.810,392.532,165.131,60.113,160.659
C06085=1013.691,-61.060,392.541,165.130,60.120,160.660
C06086=1013.685,-61.310,392.551,165.127,60.127,160.660
C06087=1013.681,-61.560,392.561,165.126,60.134,160.661
C06088=1013.676,-61.810,392.570,165.122,60.140,160.661
C06089=1013.671,-62.059,392.580,165.119,60.147,160.662
C06090=1013.667,-62.309,392.589,165.118,60.153,160.663
C06091=1013.662,-62.558,392.599,165.115,60.160,160.663
C06092=1013.657,-62.809,392.608,165.113,60.166,160.663
C06093=1013.652,-63.059,392.618,165.110,60.173,160.664
C06094=1013.647,-63.308,392.628,165.108,60.179,160.665
C06095=1013.643,-63.558,392.637,165.105,60.186,160.665
C06096=1013.638,-63.807,392.647,165.103,60.192,160.666
C06097=1013.633,-64.057,392.656,165.101,60.199,160.666
C06098=1013.628,-64.307,392.666,165.099,60.205,160.667
C06099=1013.624,-64.556,392.676,165.095,60.212,160.667
C06100=1013.618,-64.807,392.685,165.093,60.218,160.668
C06101=1013.614,-65.056,392.695,165.090,60.224,160.668
C06102=1013.610,-65.307,392.705,165.088,60.231,160.668
C06103=1013.605,-65.556,392.714,165.086,60.238,160.669
C06104=1013.600,-65.806,392.723,165.084,60.244,160.670
C06105=1013.596,-66.056,392.733,165.082,60.250,160.670
C06106=1013.591,-66.306,392.742,165.079,60.257,160.671
C06107=1013.586,-66.555,392.752,165.077,60.263,160.671
C06108=1013.582,-66.805,392.761,165.073,60.269,160.671
C06109=1013.577,-67.054,392.771,165.071,60.275,160.672
C06110=1013.572,-67.304,392.780,165.069,60.281,160.672
C06111=1013.568,-67.554,392.790,165.066,60.288,160.673
C06112=1013.563,-67.804,392.799,165.064,60.294,160.673
///RCONF 1,0,0,0,1,0,0,0,0,0,0,0,0,0,0,0,0,0,0,0,0,0,0,0
C06113=1013.558,-68.053,392.809,165.062,60.300,160.674
C06114=1013.554,-68.303,392.818,165.059,60.307,160.674
C06115=1013.549,-68.553,392.827,165.057,60.313,160.675
C06116=1013.544,-68.803,392.837,165.055,60.319,160.675
C06117=1013.539,-69.053,392.846,165.052,60.325,160.676
C06118=1013.534,-69.303,392.856,165.050,60.331,160.676
C06119=1013.530,-69.553,392.865,165.048,60.337,160.677
C06120=1013.524,-69.828,392.875,165.045,60.344,160.677
C06121=1013.520,-70.104,392.886,165.042,60.351,160.678
C06122=1013.514,-70.380,392.896,165.039,60.358,160.678
C06123=1013.510,-70.657,392.906,165.037,60.364,160.678
C06124=1013.505,-70.906,392.916,165.034,60.371,160.679
C06125=1013.500,-71.156,392.925,165.032,60.377,160.679
C06126=1013.495,-71.406,392.935,165.030,60.383,160.680
C06127=1013.491,-71.656,392.944,165.028,60.389,160.680
C06128=1013.486,-71.906,392.953,165.024,60.395,160.680
C06129=1013.481,-72.155,392.963,165.022,60.401,160.681
C06130=1013.477,-72.405,392.972,165.020,60.407,160.681
C06131=1013.472,-72.655,392.981,165.018,60.413,160.682
C06132=1013.468,-72.905,392.991,165.016,60.418,160.682
C06133=1013.463,-73.155,393.000,165.014,60.424,160.683
C06134=1013.459,-73.404,393.008,165.010,60.431,160.683
C06135=1013.454,-73.653,393.018,165.008,60.436,160.683
C06136=1013.450,-73.903,393.027,165.006,60.442,160.684
C06137=1013.445,-74.153,393.036,165.004,60.448,160.684
C06138=1013.440,-74.403,393.046,165.001,60.454,160.684
C06139=1013.436,-74.653,393.055,164.999,60.460,160.685
C06140=1013.431,-74.903,393.064,164.996,60.465,160.685
C06141=1013.427,-75.153,393.073,164.993,60.472,160.685
C06142=1013.422,-75.403,393.082,164.991,60.478,160.686
C06143=1013.417,-75.653,393.091,164.989,60.484,160.687
C06144=1013.412,-75.902,393.101,164.987,60.489,160.687
C06145=1013.408,-76.151,393.109,164.985,60.495,160.687
C06146=1013.403,-76.401,393.118,164.981,60.502,160.688
C06147=1013.398,-76.651,393.127,164.979,60.508,160.688
C06148=1013.394,-76.901,393.136,164.977,60.513,160.688
C06149=1013.389,-77.151,393.145,164.975,60.519,160.689
C06150=1013.384,-77.401,393.154,164.972,60.525,160.689
C06151=1013.380,-77.651,393.163,164.970,60.531,160.690
C06152=1013.375,-77.900,393.171,164.968,60.537,160.690
C06153=1013.370,-78.150,393.180,164.965,60.542,160.690
C06154=1013.366,-78.400,393.189,164.962,60.549,160.691
C06155=1013.361,-78.650,393.198,164.960,60.554,160.691
C06156=1013.356,-78.900,393.207,164.958,60.560,160.691
C06157=1013.352,-79.149,393.215,164.955,60.566,160.692
C06158=1013.347,-79.399,393.224,164.953,60.572,160.692
C06159=1013.342,-79.649,393.233,164.950,60.577,160.692
C06160=1013.338,-79.899,393.242,164.948,60.583,160.693
C06161=1013.333,-80.149,393.251,164.945,60.589,160.693
C06162=1013.328,-80.399,393.260,164.944,60.595,160.694
C06163=1013.324,-80.649,393.269,164.941,60.600,160.694
C06164=1013.319,-80.898,393.277,164.939,60.606,160.694
C06165=1013.315,-81.148,393.285,164.936,60.612,160.695
C06166=1013.309,-81.398,393.294,164.934,60.618,160.695
C06167=1013.305,-81.648,393.303,164.932,60.624,160.696
C06168=1013.300,-81.897,393.311,164.929,60.629,160.696
C06169=1013.295,-82.147,393.319,164.926,60.636,160.696
C06170=1013.291,-82.397,393.328,164.924,60.641,160.696
C06171=1013.285,-82.647,393.336,164.922,60.647,160.697
C06172=1013.282,-82.896,393.345,164.919,60.653,160.697
C06173=1013.276,-83.146,393.353,164.917,60.659,160.698
C06174=1013.272,-83.397,393.362,164.914,60.664,160.698
C06175=1013.267,-83.646,393.370,164.912,60.669,160.698
C06176=1013.262,-83.896,393.378,164.910,60.676,160.698
C06177=1013.258,-84.146,393.387,164.907,60.681,160.699
C06178=1013.253,-84.396,393.395,164.905,60.687,160.699
C06179=1013.249,-84.645,393.404,164.902,60.692,160.699
C06180=1013.243,-84.895,393.412,164.900,60.698,160.700
C06181=1013.238,-85.145,393.421,164.899,60.703,160.700
C06182=1013.235,-85.395,393.429,164.896,60.709,160.701
C06183=1013.229,-85.644,393.437,164.893,60.714,160.701
C06184=1013.225,-85.922,393.447,164.890,60.721,160.701
C06185=1013.219,-86.200,393.456,164.888,60.727,160.702
C06186=1013.214,-86.479,393.465,164.885,60.733,160.701
C06187=1013.209,-86.756,393.474,164.883,60.739,160.702
C06188=1013.205,-87.006,393.483,164.880,60.744,160.702
C06189=1013.199,-87.256,393.492,164.877,60.750,160.702
C06190=1013.195,-87.505,393.499,164.875,60.756,160.703
C06191=1013.190,-87.755,393.508,164.874,60.761,160.703
C06192=1013.185,-88.005,393.517,164.871,60.766,160.704
C06193=1013.181,-88.255,393.525,164.868,60.771,160.704
C06194=1013.176,-88.505,393.533,164.866,60.777,160.704
C06195=1013.172,-88.754,393.541,164.863,60.782,160.704
C06196=1013.167,-89.005,393.550,164.861,60.787,160.705
C06197=1013.162,-89.254,393.558,164.859,60.792,160.705
C06198=1013.158,-89.504,393.566,164.856,60.798,160.705
C06199=1013.153,-89.754,393.575,164.853,60.803,160.705
C06200=1013.149,-90.004,393.582,164.852,60.808,160.706
C06201=1013.144,-90.254,393.591,164.849,60.813,160.706
C06202=1013.139,-90.503,393.600,164.846,60.819,160.706
C06203=1013.135,-90.753,393.608,164.844,60.824,160.706
C06204=1013.130,-91.003,393.616,164.842,60.829,160.706
C06205=1013.126,-91.253,393.624,164.840,60.834,160.707
C06206=1013.121,-91.503,393.633,164.837,60.840,160.707
C06207=1013.117,-91.752,393.640,164.835,60.845,160.707
C06208=1013.112,-92.002,393.649,164.833,60.850,160.707
C06209=1013.107,-92.253,393.657,164.830,60.855,160.708
C06210=1013.104,-92.502,393.666,164.828,60.860,160.708
C06211=1013.099,-92.752,393.673,164.826,60.866,160.708
C06212=1013.094,-93.001,393.682,164.823,60.870,160.708
C06213=1013.090,-93.252,393.690,164.821,60.875,160.709
C06214=1013.085,-93.501,393.698,164.818,60.881,160.709
C06215=1013.081,-93.752,393.706,164.817,60.886,160.709
C06216=1013.076,-94.001,393.714,164.813,60.890,160.709
C06217=1013.071,-94.251,393.722,164.812,60.895,160.709
C06218=1013.067,-94.500,393.731,164.809,60.900,160.710
C06219=1013.062,-94.751,393.739,164.807,60.905,160.710
C06220=1013.058,-95.000,393.747,164.804,60.910,160.710
C06221=1013.053,-95.250,393.755,164.802,60.915,160.710
C06222=1013.049,-95.499,393.763,164.800,60.920,160.710
C06223=1013.045,-95.750,393.772,164.797,60.924,160.710
C06224=1013.040,-95.999,393.780,164.795,60.930,160.711
C06225=1013.035,-96.249,393.788,164.793,60.935,160.711
C06226=1013.031,-96.499,393.796,164.790,60.939,160.711
C06227=1013.026,-96.749,393.804,164.788,60.944,160.711
C06228=1013.022,-96.999,393.812,164.785,60.949,160.711
C06229=1013.018,-97.248,393.820,164.783,60.954,160.712
C06230=1013.013,-97.498,393.828,164.781,60.958,160.712
C06231=1013.009,-97.748,393.836,164.778,60.963,160.712
C06232=1013.004,-97.998,393.844,164.776,60.968,160.712
C06233=1013.000,-98.247,393.852,164.773,60.973,160.712
C06234=1012.995,-98.498,393.860,164.772,60.978,160.712
C06235=1012.991,-98.748,393.868,164.769,60.982,160.712
C06236=1012.986,-98.997,393.876,164.767,60.987,160.713
C06237=1012.981,-99.247,393.884,164.764,60.992,160.712
C06238=1012.977,-99.497,393.891,164.762,60.997,160.713
C06239=1012.972,-99.747,393.899,164.760,61.002,160.713
C06240=1012.968,-99.997,393.906,164.757,61.006,160.713
C06241=1012.963,-100.247,393.914,164.756,61.011,160.714
C06242=1012.959,-100.496,393.923,164.752,61.016,160.713
C06243=1012.954,-100.746,393.930,164.751,61.021,160.714
C06244=1012.949,-100.996,393.938,164.748,61.025,160.714
C06245=1012.945,-101.246,393.945,164.746,61.031,160.714
C06246=1012.941,-101.496,393.953,164.743,61.035,160.714
C06247=1012.936,-101.746,393.960,164.741,61.039,160.714
C06248=1012.931,-102.039,393.969,164.738,61.044,160.714
C06249=1012.925,-102.333,393.978,164.736,61.050,160.715
C06250=1012.920,-102.626,393.987,164.732,61.055,160.714
C06251=1012.915,-102.920,393.997,164.729,61.061,160.715
C06252=1012.910,-103.170,394.005,164.728,61.066,160.715
C06253=1012.906,-103.420,394.012,164.726,61.070,160.715
C06254=1012.902,-103.669,394.019,164.723,61.074,160.715
C06255=1012.897,-103.919,394.027,164.721,61.080,160.715
C06256=1012.892,-104.169,394.035,164.718,61.084,160.715
C06257=1012.888,-104.419,394.042,164.716,61.088,160.715
C06258=1012.883,-104.669,394.050,164.714,61.092,160.716
C06259=1012.879,-104.919,394.057,164.712,61.097,160.716
C06260=1012.874,-105.168,394.064,164.709,61.102,160.716
C06261=1012.870,-105.419,394.073,164.707,61.106,160.716
C06262=1012.866,-105.669,394.080,164.704,61.110,160.716
C06263=1012.861,-105.918,394.088,164.702,61.114,160.716
C06264=1012.857,-106.168,394.095,164.700,61.118,160.716
C06265=1012.852,-106.418,394.103,164.698,61.123,160.716
C06266=1012.848,-106.668,394.110,164.696,61.127,160.717
C06267=1012.843,-106.918,394.118,164.693,61.132,160.716
C06268=1012.844,-94.477,393.307,164.795,61.158,160.755
C06269=1012.847,-94.228,393.298,164.797,61.153,160.754
C06270=1012.852,-93.977,393.290,164.799,61.149,160.754
C06271=1012.856,-93.728,393.282,164.801,61.145,160.754
C06272=1012.861,-93.478,393.274,164.804,61.139,160.754
C06273=1012.866,-93.229,393.266,164.806,61.135,160.754
C06274=1012.870,-92.978,393.257,164.808,61.130,160.754
C06275=1012.875,-92.729,393.249,164.811,61.126,160.754
C06276=1012.879,-92.478,393.241,164.813,61.121,160.754
C06277=1012.884,-92.229,393.233,164.815,61.116,160.753
C06278=1012.889,-91.979,393.225,164.818,61.112,160.754
C06279=1012.893,-91.730,393.216,164.820,61.107,160.753
C06280=1012.898,-91.479,393.209,164.822,61.103,160.753
C06281=1012.901,-91.230,393.200,164.825,61.097,160.753
C06282=1012.906,-90.980,393.192,164.826,61.092,160.752
C06283=1012.911,-90.731,393.184,164.830,61.088,160.753
C06284=1012.915,-90.480,393.176,164.831,61.083,160.752
C06285=1012.920,-90.231,393.167,164.835,61.078,160.752
C06286=1012.924,-89.980,393.159,164.836,61.073,160.752
C06287=1012.929,-89.731,393.151,164.839,61.068,160.752
C06288=1012.934,-89.481,393.143,164.841,61.064,160.752
C06289=1012.938,-89.231,393.134,164.844,61.058,160.751
C06290=1012.943,-88.982,393.126,164.845,61.053,160.751
C06291=1012.947,-88.731,393.118,164.849,61.049,160.751
C06292=1012.952,-88.482,393.110,164.850,61.044,160.751
C06293=1012.957,-88.232,393.102,164.853,61.038,160.750
C06294=1012.961,-87.982,393.093,164.854,61.034,160.750
C06295=1012.966,-87.732,393.085,164.858,61.029,160.750
C06296=1012.970,-87.482,393.076,164.859,61.024,160.750
C06297=1012.974,-87.256,393.068,164.861,61.019,160.749
C06298=1012.979,-87.030,393.062,164.864,61.014,160.750
C06299=1012.983,-86.804,393.054,164.866,61.010,160.749
C06300=1012.987,-86.578,393.046,164.868,61.005,160.749
C06301=1012.991,-86.352,393.038,164.870,61.000,160.749
C06302=1012.995,-86.125,393.031,164.872,60.996,160.748
C06303=1013.000,-85.899,393.024,164.874,60.991,160.748
C06304=1013.004,-85.673,393.016,164.877,60.987,160.748
C06305=1013.008,-85.422,393.008,164.878,60.982,160.748
C06306=1013.013,-85.173,393.000,164.881,60.976,160.748
C06307=1013.017,-84.923,392.991,164.884,60.971,160.747
C06308=1013.022,-84.673,392.983,164.886,60.966,160.747
C06309=1013.027,-84.424,392.975,164.888,60.961,160.747
C06310=1013.032,-84.174,392.966,164.890,60.955,160.747
C06311=1013.037,-83.924,392.957,164.893,60.950,160.746
C06312=1013.040,-83.674,392.949,164.895,60.945,160.746
C06313=1013.046,-83.425,392.941,164.897,60.940,160.746
C06314=1013.051,-83.175,392.932,164.900,60.934,160.746
C06315=1013.055,-82.924,392.924,164.903,60.929,160.745
C06316=1013.060,-82.675,392.916,164.905,60.924,160.745
C06317=1013.064,-82.425,392.907,164.906,60.918,160.744
C06318=1013.070,-82.175,392.898,164.909,60.912,160.744
C06319=1013.073,-81.926,392.890,164.911,60.907,160.744
C06320=1013.079,-81.676,392.882,164.914,60.902,160.744
C06321=1013.084,-81.426,392.873,164.917,60.896,160.744
C06322=1013.088,-81.176,392.864,164.917,60.891,160.743
C06323=1013.093,-80.926,392.857,164.920,60.885,160.743
C06324=1013.097,-80.676,392.848,164.923,60.880,160.742
C06325=1013.102,-80.427,392.839,164.925,60.875,160.742
C06326=1013.107,-80.177,392.830,164.928,60.869,160.742
C06327=1013.111,-79.927,392.821,164.930,60.863,160.741
C06328=1013.116,-79.678,392.813,164.932,60.858,160.741
C06329=1013.121,-79.428,392.804,164.934,60.853,160.741
C06330=1013.125,-79.178,392.795,164.937,60.847,160.741
C06331=1013.129,-78.927,392.786,164.940,60.842,160.740
C06332=1013.134,-78.678,392.778,164.942,60.837,160.740
C06333=1013.139,-78.428,392.769,164.944,60.831,160.740
C06334=1013.143,-78.178,392.760,164.947,60.825,160.739
C06335=1013.148,-77.928,392.752,164.948,60.820,160.739
C06336=1013.153,-77.678,392.743,164.951,60.815,160.739
C06337=1013.157,-77.429,392.734,164.953,60.809,160.738
C06338=1013.162,-77.179,392.725,164.956,60.803,160.738
C06339=1013.167,-76.929,392.716,164.958,60.798,160.738
C06340=1013.172,-76.680,392.706,164.960,60.792,160.737
C06341=1013.176,-76.430,392.697,164.963,60.787,160.737
C06342=1013.181,-76.180,392.689,164.965,60.780,160.737
C06343=1013.185,-75.931,392.680,164.968,60.775,160.736
C06344=1013.190,-75.681,392.671,164.970,60.770,160.736
C06345=1013.195,-75.431,392.663,164.972,60.764,160.736
C06346=1013.200,-75.181,392.654,164.975,60.758,160.735
C06347=1013.204,-74.931,392.644,164.977,60.752,160.735
C06348=1013.209,-74.681,392.635,164.980,60.747,160.735
C06349=1013.213,-74.431,392.626,164.982,60.741,160.734
C06350=1013.217,-74.182,392.617,164.984,60.735,160.734
C06351=1013.222,-73.932,392.608,164.987,60.730,160.734
C06352=1013.226,-73.682,392.599,164.988,60.725,160.733
C06353=1013.231,-73.432,392.590,164.990,60.719,160.733
C06354=1013.236,-73.183,392.580,164.993,60.713,160.732
C06355=1013.240,-72.933,392.571,164.995,60.707,160.732
C06356=1013.245,-72.682,392.562,164.998,60.702,160.732
C06357=1013.250,-72.433,392.552,165.000,60.697,160.732
C06358=1013.254,-72.183,392.543,165.002,60.690,160.731
C06359=1013.259,-71.933,392.534,165.005,60.685,160.731
C06360=1013.263,-71.684,392.524,165.007,60.679,160.730
C06361=1013.267,-71.434,392.515,165.010,60.674,160.730
C06362=1013.272,-71.184,392.506,165.012,60.668,160.729
C06363=1013.277,-70.935,392.496,165.014,60.662,160.729
C06364=1013.281,-70.685,392.487,165.016,60.656,160.729
C06365=1013.287,-70.409,392.477,165.019,60.649,160.728
C06366=1013.292,-70.133,392.466,165.022,60.643,160.728
C06367=1013.297,-69.857,392.457,165.024,60.637,160.728
C06368=1013.302,-69.581,392.446,165.027,60.630,160.727
C06369=1013.307,-69.331,392.436,165.029,60.624,160.727
C06370=1013.311,-69.081,392.427,165.032,60.619,160.726
C06371=1013.316,-68.831,392.418,165.034,60.613,160.726
C06372=1013.320,-68.582,392.408,165.036,60.607,160.725
C06373=1013.325,-68.332,392.399,165.038,60.600,160.725
C06374=1013.330,-68.083,392.389,165.042,60.595,160.725
C06375=1013.334,-67.833,392.380,165.044,60.588,160.724
C06376=1013.339,-67.583,392.371,165.046,60.582,160.724
C06377=1013.344,-67.333,392.362,165.048,60.577,160.724
C06378=1013.348,-67.083,392.352,165.050,60.571,160.723
C06379=1013.353,-66.834,392.343,165.052,60.565,160.722
C06380=1013.358,-66.584,392.334,165.055,60.558,160.722
///RCONF 1,0,0,0,0,0,0,0,0,0,0,0,0,0,0,0,0,0,0,0,0,0,0,0
C06381=1013.362,-66.334,392.324,165.057,60.552,160.722
C06382=1013.367,-66.084,392.315,165.060,60.547,160.721
C06383=1013.372,-65.835,392.305,165.062,60.541,160.721
C06384=1013.376,-65.585,392.296,165.065,60.534,160.720
C06385=1013.381,-65.335,392.286,165.067,60.528,160.720
C06386=1013.386,-65.085,392.277,165.069,60.522,160.719
C06387=1013.390,-64.836,392.267,165.071,60.516,160.719
C06388=1013.395,-64.586,392.258,165.074,60.509,160.718
C06389=1013.400,-64.337,392.248,165.076,60.503,160.718
C06390=1013.404,-64.087,392.239,165.078,60.497,160.717
C06391=1013.409,-63.837,392.229,165.081,60.491,160.717
C06392=1013.414,-63.586,392.220,165.083,60.484,160.716
C06393=1013.419,-63.337,392.210,165.085,60.478,160.716
C06394=1013.424,-63.087,392.201,165.088,60.472,160.716
C06395=1013.428,-62.838,392.191,165.090,60.466,160.715
C06396=1013.433,-62.587,392.182,165.092,60.460,160.714
C06397=1013.438,-62.338,392.172,165.095,60.453,160.714
C06398=1013.442,-62.088,392.163,165.097,60.447,160.714
C06399=1013.447,-61.839,392.154,165.100,60.440,160.713
C06400=1013.452,-61.589,392.144,165.102,60.434,160.713
C06401=1013.457,-61.339,392.134,165.104,60.428,160.712
C06402=1013.462,-61.089,392.124,165.108,60.422,160.712
C06403=1013.467,-60.839,392.115,165.109,60.415,160.711
C06404=1013.471,-60.590,392.106,165.112,60.408,160.711
C06405=1013.476,-60.340,392.096,165.114,60.402,160.710
C06406=1013.481,-60.090,392.087,165.117,60.396,160.710
C06407=1013.485,-59.841,392.076,165.119,60.390,160.709
C06408=1013.490,-59.590,392.067,165.121,60.382,160.708
C06409=1013.495,-59.340,392.057,165.123,60.376,160.708
C06410=1013.500,-59.091,392.047,165.127,60.370,160.708
C06411=1013.504,-58.841,392.038,165.129,60.363,160.707
C06412=1013.509,-58.592,392.028,165.131,60.356,160.706
C06413=1013.514,-58.342,392.019,165.133,60.350,160.706
C06414=1013.519,-58.091,392.009,165.136,60.344,160.706
C06415=1013.524,-57.842,391.999,165.137,60.337,160.705
C06416=1013.529,-57.593,391.990,165.140,60.330,160.704
C06417=1013.533,-57.343,391.981,165.142,60.324,160.704
C06418=1013.538,-57.093,391.971,165.145,60.317,160.703
C06419=1013.543,-56.843,391.961,165.147,60.311,160.702
C06420=1013.548,-56.593,391.951,165.149,60.303,160.702
C06421=1013.553,-56.344,391.942,165.152,60.297,160.701
C06422=1013.558,-56.094,391.932,165.154,60.291,160.701
C06423=1013.563,-55.844,391.922,165.157,60.283,160.700
C06424=1013.568,-55.594,391.913,165.160,60.277,160.700
C06425=1013.572,-55.345,391.903,165.161,60.270,160.699
C06426=1013.577,-55.095,391.893,165.164,60.264,160.699
C06427=1013.583,-54.845,391.883,165.166,60.257,160.698
C06428=1013.587,-54.595,391.874,165.169,60.250,160.697
C06429=1013.592,-54.320,391.862,165.171,60.242,160.696
C06430=1013.597,-54.046,391.852,165.174,60.234,160.696
C06431=1013.603,-53.771,391.841,165.176,60.227,160.695
C06432=1013.609,-53.496,391.830,165.179,60.220,160.695
C06433=1013.613,-53.247,391.821,165.181,60.213,160.694
C06434=1013.619,-52.996,391.811,165.184,60.206,160.694
C06435=1013.623,-52.747,391.801,165.186,60.199,160.693
C06436=1013.628,-52.497,391.792,165.188,60.192,160.692
C06437=1013.633,-52.248,391.782,165.191,60.185,160.692
C06438=1013.638,-51.998,391.772,165.194,60.178,160.691
C06439=1013.643,-51.748,391.763,165.195,60.171,160.690
C06440=1013.648,-51.498,391.753,165.198,60.165,160.690
C06441=1013.653,-51.248,391.742,165.201,60.158,160.689
C06442=1013.657,-50.998,391.732,165.203,60.150,160.689
C06443=1013.662,-50.748,391.721,165.205,60.144,160.688
C06444=1013.667,-50.498,391.712,165.208,60.137,160.687
C06445=1013.671,-50.249,391.701,165.210,60.131,160.687
C06446=1013.676,-49.999,391.691,165.212,60.124,160.686
C06447=1013.681,-49.749,391.681,165.215,60.117,160.686
C06448=1013.686,-49.499,391.671,165.216,60.110,160.685
C06449=1013.691,-49.250,391.660,165.219,60.103,160.684
C06450=1013.695,-49.000,391.650,165.222,60.096,160.684
C06451=1013.701,-48.750,391.639,165.223,60.090,160.683
C06452=1013.705,-48.501,391.629,165.227,60.083,160.683
C06453=1013.710,-48.251,391.619,165.229,60.076,160.682
C06454=1013.714,-48.001,391.609,165.231,60.069,160.681
C06455=1013.719,-47.751,391.599,165.233,60.062,160.681
C06456=1013.724,-47.501,391.588,165.236,60.055,160.680
C06457=1013.729,-47.252,391.577,165.238,60.048,160.679
C06458=1013.734,-47.003,391.568,165.241,60.041,160.679
C06459=1013.738,-46.752,391.557,165.243,60.035,160.678
C06460=1013.743,-46.503,391.547,165.245,60.027,160.678
C06461=1013.748,-46.252,391.536,165.248,60.020,160.677
C06462=1013.753,-46.004,391.526,165.250,60.013,160.676
C06463=1013.758,-45.753,391.515,165.252,60.007,160.676
C06464=1013.763,-45.504,391.505,165.255,60.000,160.675
C06465=1013.767,-45.254,391.495,165.257,59.992,160.674
C06466=1013.772,-45.004,391.485,165.260,59.985,160.674
C06467=1013.777,-44.755,391.474,165.262,59.978,160.673
C06468=1013.782,-44.505,391.463,165.263,59.971,160.672
C06469=1013.786,-44.255,391.453,165.267,59.964,160.672
C06470=1013.791,-44.005,391.443,165.269,59.957,160.671
C06471=1013.796,-43.756,391.432,165.272,59.950,160.670
C06472=1013.801,-43.506,391.422,165.274,59.943,160.670
C06473=1013.806,-43.256,391.412,165.276,59.935,160.669
C06474=1013.811,-43.006,391.401,165.279,59.928,160.668
C06475=1013.816,-42.757,391.391,165.280,59.921,160.667
C06476=1013.821,-42.507,391.380,165.283,59.914,160.667
C06477=1013.826,-42.257,391.370,165.285,59.907,160.666
C06478=1013.830,-42.007,391.359,165.288,59.900,160.665
C06479=1013.835,-41.758,391.349,165.290,59.892,160.665
C06480=1013.840,-41.508,391.338,165.293,59.885,160.664
C06481=1013.845,-41.258,391.328,165.295,59.878,160.663
C06482=1013.850,-41.008,391.317,165.298,59.871,160.663
C06483=1013.855,-40.759,391.307,165.300,59.863,160.662
C06484=1013.859,-40.509,391.296,165.303,59.856,160.661
C06485=1013.865,-40.260,391.286,165.304,59.848,160.660
C06486=1013.869,-40.009,391.275,165.307,59.841,160.660
C06487=1013.874,-39.760,391.265,165.309,59.834,160.659
C06488=1013.879,-39.510,391.254,165.312,59.826,160.658
C06489=1013.884,-39.260,391.244,165.314,59.819,160.658
C06490=1013.889,-39.011,391.232,165.317,59.812,160.657
C06491=1013.894,-38.761,391.222,165.318,59.805,160.656
C06492=1013.898,-38.511,391.211,165.321,59.798,160.656
C06493=1013.903,-38.237,391.198,165.324,59.789,160.655
C06494=1013.909,-37.962,391.188,165.326,59.782,160.654
C06495=1013.914,-37.687,391.176,165.329,59.774,160.653
C06496=1013.919,-37.413,391.163,165.331,59.766,160.652
C06497=1013.924,-37.163,391.152,165.333,59.759,160.652
C06498=1013.929,-36.913,391.142,165.336,59.751,160.651
C06499=1013.934,-36.664,391.131,165.338,59.744,160.650
C06500=1013.939,-36.414,391.120,165.341,59.737,160.650
C06501=1013.943,-36.164,391.109,165.343,59.730,160.649
C06502=1013.948,-35.915,391.097,165.346,59.722,160.648
C06503=1013.953,-35.665,391.088,165.348,59.714,160.647
C06504=1013.958,-35.415,391.076,165.350,59.707,160.647
C06505=1013.963,-35.165,391.065,165.353,59.700,160.646
C06506=1013.967,-34.916,391.054,165.355,59.693,160.645
C06507=1013.973,-34.666,391.043,165.358,59.686,160.645
C06508=1013.978,-34.416,391.033,165.359,59.678,160.644
C06509=1013.982,-34.167,391.022,165.362,59.670,160.643
C06510=1013.987,-33.916,391.011,165.364,59.663,160.642
C06511=1013.993,-33.667,391.000,165.366,59.655,160.641
C06512=1013.997,-33.418,390.989,165.369,59.648,160.641
C06513=1014.002,-33.167,390.978,165.371,59.641,160.640
C06514=1014.007,-32.918,390.967,165.374,59.632,160.639
C06515=1014.012,-32.669,390.956,165.377,59.625,160.639
C06516=1014.017,-32.418,390.945,165.379,59.618,160.638
C06517=1014.022,-32.169,390.934,165.381,59.610,160.637
C06518=1014.026,-31.920,390.923,165.384,59.603,160.636
C06519=1014.031,-31.669,390.912,165.386,59.595,160.636
C06520=1014.036,-31.420,390.901,165.388,59.587,160.635
C06521=1014.041,-31.170,390.890,165.391,59.580,160.634
C06522=1014.046,-30.921,390.878,165.392,59.572,160.633
C06523=1014.050,-30.670,390.868,165.396,59.565,160.632
C06524=1014.056,-30.421,390.857,165.398,59.557,160.631
C06525=1014.061,-30.172,390.846,165.400,59.549,160.631
C06526=1014.065,-29.921,390.835,165.402,59.542,160.630
C06527=1014.070,-29.671,390.824,165.405,59.534,160.629
C06528=1014.076,-29.422,390.813,165.407,59.526,160.628
C06529=1014.080,-29.173,390.802,165.410,59.519,160.628
C06530=1014.085,-28.922,390.791,165.412,59.511,160.627
C06531=1014.090,-28.673,390.779,165.415,59.504,160.626
C06532=1014.096,-28.423,390.768,165.417,59.496,160.625
C06533=1014.100,-28.174,390.757,165.418,59.488,160.624
C06534=1014.105,-27.924,390.747,165.422,59.480,160.624
C06535=1014.110,-27.674,390.735,165.424,59.472,160.623
C06536=1014.115,-27.424,390.724,165.426,59.465,160.622
C06537=1014.120,-27.174,390.712,165.428,59.457,160.621
C06538=1014.125,-26.924,390.701,165.431,59.450,160.620
C06539=1014.129,-26.675,390.690,165.433,59.442,160.620
C06540=1014.134,-26.426,390.678,165.435,59.435,160.619
C06541=1014.139,-26.176,390.667,165.438,59.427,160.618
C06542=1014.144,-25.926,390.655,165.441,59.419,160.617
C06543=1014.149,-25.676,390.644,165.443,59.411,160.616
C06544=1014.154,-25.427,390.633,165.445,59.404,160.616
C06545=1014.159,-25.177,390.621,165.447,59.396,160.615
C06546=1014.163,-24.927,390.609,165.450,59.389,160.614
C06547=1014.168,-24.677,390.598,165.452,59.381,160.613
C06548=1014.173,-24.428,390.586,165.455,59.373,160.612
C06549=1014.178,-24.178,390.575,165.457,59.365,160.611
C06550=1014.182,-23.929,390.564,165.459,59.357,160.610
C06551=1014.187,-23.679,390.552,165.462,59.350,160.610
C06552=1014.192,-23.429,390.541,165.463,59.342,160.609
C06553=1014.197,-23.179,390.529,165.466,59.334,160.608
C06554=1014.202,-22.929,390.518,165.469,59.327,160.607
C06555=1014.207,-22.680,390.506,165.471,59.319,160.606
C06556=1014.212,-22.430,390.495,165.473,59.311,160.605
C06557=1014.218,-22.154,390.482,165.476,59.302,160.605
C06558=1014.223,-21.879,390.469,165.478,59.293,160.604
C06559=1014.229,-21.603,390.456,165.481,59.285,160.603
C06560=1014.234,-21.328,390.444,165.484,59.276,160.602
C06561=1014.239,-21.078,390.432,165.486,59.268,160.601
C06562=1014.244,-20.828,390.420,165.489,59.260,160.600
C06563=1014.249,-20.578,390.409,165.491,59.252,160.599
C06564=1014.254,-20.329,390.397,165.493,59.244,160.598
C06565=1014.258,-20.080,390.386,165.497,59.237,160.598
C06566=1014.263,-19.830,390.375,165.498,59.229,160.597
C06567=1014.268,-19.580,390.363,165.500,59.221,160.596
C06568=1014.273,-19.331,390.351,165.503,59.212,160.595
C06569=1014.278,-19.081,390.339,165.505,59.204,160.594
C06570=1014.283,-18.831,390.328,165.507,59.197,160.593
C06571=1014.288,-18.581,390.316,165.510,59.188,160.592
C06572=1014.293,-18.332,390.305,165.512,59.180,160.591
C06573=1014.298,-18.082,390.294,165.514,59.172,160.590
C06574=1014.304,-17.833,390.281,165.517,59.164,160.590
C06575=1014.309,-17.583,390.270,165.520,59.157,160.589
C06576=1014.314,-17.333,390.258,165.522,59.149,160.588
C06577=1014.319,-17.083,390.247,165.525,59.141,160.587
C06578=1014.324,-16.833,390.235,165.527,59.133,160.586
C06579=1014.328,-16.584,390.223,165.530,59.124,160.585
C06580=1014.333,-16.334,390.211,165.532,59.116,160.584
C06581=1014.338,-16.084,390.200,165.533,59.108,160.583
C06582=1014.343,-15.834,390.188,165.537,59.100,160.583
C06583=1014.348,-15.585,390.175,165.538,59.092,160.582
C06584=1014.353,-15.335,390.164,165.540,59.084,160.581
C06585=1014.358,-15.085,390.153,165.543,59.076,160.580
C06586=1014.362,-14.836,390.140,165.545,59.068,160.579
C06587=1014.367,-14.586,390.128,165.547,59.060,160.578
C06588=1014.373,-14.337,390.116,165.550,59.052,160.577
C06589=1014.377,-14.087,390.104,165.552,59.044,160.576
C06590=1014.382,-13.837,390.093,165.554,59.036,160.575
C06591=1014.387,-13.588,390.080,165.558,59.028,160.575
C06592=1014.392,-13.338,390.068,165.560,59.021,160.574
C06593=1014.397,-13.088,390.056,165.562,59.013,160.573
C06594=1014.402,-12.839,390.045,165.565,59.004,160.572
C06595=1014.406,-12.589,390.032,165.567,58.996,160.571
C06596=1014.411,-12.339,390.020,165.570,58.988,160.570
C06597=1014.416,-12.090,390.009,165.571,58.979,160.569
C06598=1014.421,-11.840,389.996,165.573,58.972,160.568
C06599=1014.427,-11.590,389.984,165.576,58.963,160.567
C06600=1014.432,-11.340,389.972,165.578,58.955,160.566
C06601=1014.436,-11.090,389.960,165.581,58.947,160.566
C06602=1014.441,-10.841,389.948,165.583,58.939,160.565
C06603=1014.446,-10.591,389.936,165.585,58.931,160.564
C06604=1014.451,-10.342,389.924,165.588,58.923,160.563
C06605=1014.456,-10.092,389.912,165.590,58.915,160.562
C06606=1014.461,-9.843,389.899,165.593,58.907,160.561
C06607=1014.466,-9.593,389.888,165.595,58.898,160.560
C06608=1014.471,-9.344,389.876,165.598,58.890,160.559
C06609=1014.475,-9.093,389.864,165.600,58.882,160.558
C06610=1014.481,-8.844,389.851,165.603,58.874,160.557
C06611=1014.486,-8.594,389.839,165.605,58.866,160.556
C06612=1014.491,-8.344,389.827,165.607,58.857,160.555
C06613=1014.496,-8.095,389.815,165.609,58.849,160.554
C06614=1014.501,-7.845,389.803,165.611,58.841,160.553
C06615=1014.506,-7.596,389.790,165.614,58.833,160.553
C06616=1014.511,-7.346,389.779,165.617,58.823,160.551
C06617=1014.516,-7.097,389.767,165.619,58.816,160.550
C06618=1014.521,-6.847,389.754,165.622,58.807,160.550
C06619=1014.526,-6.597,389.742,165.623,58.799,160.548
C06620=1014.531,-6.348,389.730,165.626,58.790,160.548
C06621=1014.537,-6.070,389.716,165.629,58.781,160.547
C06622=1014.541,-5.792,389.703,165.631,58.772,160.545
C06623=1014.548,-5.515,389.689,165.634,58.763,160.544
C06624=1014.553,-5.237,389.675,165.636,58.753,160.543
C06625=1014.558,-4.988,389.663,165.638,58.745,160.542
C06626=1014.563,-4.739,389.652,165.642,58.737,160.541
C06627=1014.568,-4.488,389.639,165.643,58.728,160.540
C06628=1014.573,-4.239,389.626,165.646,58.720,160.539
C06629=1014.578,-3.989,389.614,165.648,58.712,160.538
C06630=1014.582,-3.740,389.602,165.651,58.704,160.538
C06631=1014.588,-3.489,389.588,165.653,58.696,160.537
C06632=1014.593,-3.240,389.576,165.655,58.687,160.535
C06633=1014.597,-2.991,389.563,165.658,58.679,160.535
C06634=1014.602,-2.741,389.551,165.660,58.671,160.534
C06635=1014.607,-2.492,389.538,165.663,58.663,160.533
C06636=1014.613,-2.242,389.525,165.664,58.654,160.532
C06637=1014.617,-1.992,389.513,165.667,58.646,160.531
C06638=1014.621,-1.742,389.501,165.669,58.638,160.530
C06639=1014.626,-1.493,389.488,165.672,58.630,160.529
C06640=1014.632,-1.243,389.475,165.674,58.621,160.528
C06641=1014.636,-0.993,389.462,165.677,58.613,160.527
C06642=1014.641,-0.744,389.450,165.679,58.605,160.526
C06643=1014.646,-0.495,389.437,165.681,58.596,160.525
C06644=1014.651,-0.244,389.424,165.684,58.588,160.524
C06645=1014.656,0.005,389.411,165.687,58.580,160.523
C06646=1014.661,0.255,389.399,165.688,58.571,160.522
C06647=1014.666,0.504,389.387,165.691,58.563,160.521
C06648=1014.671,0.754,389.373,165.693,58.554,160.520
C06649=1014.676,1.003,389.361,165.696,58.546,160.519
C06650=1014.680,1.253,389.348,165.698,58.538,160.518
C06651=1014.686,1.503,389.335,165.700,58.529,160.517
C06652=1014.691,1.752,389.322,165.702,58.521,160.516
C06653=1014.695,2.002,389.310,165.705,58.512,160.515
C06654=1014.700,2.251,389.297,165.707,58.505,160.514
C06655=1014.706,2.501,389.284,165.709,58.496,160.513
C06656=1014.710,2.751,389.272,165.711,58.488,160.512
C06657=1014.715,3.000,389.259,165.714,58.479,160.511
C06658=1014.721,3.250,389.246,165.717,58.470,160.510
C06659=1014.725,3.500,389.233,165.719,58.462,160.509
C06660=1014.730,3.749,389.221,165.722,58.454,160.508
C06661=1014.735,3.999,389.208,165.723,58.445,160.507
C06662=1014.740,4.248,389.195,165.726,58.437,160.506
C06663=1014.745,4.498,389.183,165.729,58.428,160.505
C06664=1014.750,4.748,389.169,165.731,58.420,160.504
C06665=1014.755,4.998,389.157,165.733,58.411,160.503
C06666=1014.760,5.247,389.144,165.735,58.402,160.502
C06667=1014.765,5.497,389.131,165.738,58.394,160.501
C06668=1014.770,5.746,389.118,165.740,58.385,160.500
C06669=1014.774,5.996,389.106,165.743,58.377,160.499
C06670=1014.780,6.246,389.093,165.745,58.368,160.498
C06671=1014.785,6.495,389.080,165.748,58.359,160.497
C06672=1014.790,6.746,389.067,165.750,58.351,160.496
C06673=1014.795,6.995,389.054,165.752,58.342,160.495
C06674=1014.800,7.244,389.042,165.755,58.333,160.494
C06675=1014.805,7.494,389.028,165.757,58.326,160.493
C06676=1014.810,7.743,389.016,165.759,58.317,160.492
C06677=1014.815,7.993,389.002,165.762,58.308,160.491
C06678=1014.820,8.243,388.990,165.763,58.299,160.490
C06679=1014.825,8.492,388.977,165.767,58.291,160.489
C06680=1014.830,8.742,388.964,165.769,58.282,160.488
C06681=1014.835,8.992,388.952,165.771,58.273,160.487
C06682=1014.841,9.241,388.938,165.773,58.264,160.486
C06683=1014.845,9.491,388.926,165.776,58.255,160.484
C06684=1014.850,9.740,388.913,165.779,58.247,160.484
C06685=1014.856,10.019,388.898,165.781,58.237,160.482
C06686=1014.862,10.300,388.884,165.784,58.227,160.481
C06687=1014.868,10.579,388.869,165.786,58.218,160.480
C06688=1014.873,10.858,388.854,165.790,58.208,160.479
C06689=1014.879,11.108,388.842,165.792,58.199,160.478
C06690=1014.883,11.358,388.829,165.794,58.191,160.477
C06691=1014.888,11.608,388.816,165.796,58.182,160.476
C06692=1014.893,11.857,388.803,165.799,58.173,160.474
C06693=1014.899,12.107,388.790,165.801,58.164,160.473
C06694=1014.904,12.356,388.777,165.803,58.155,160.472
C06695=1014.909,12.606,388.764,165.805,58.146,160.471
C06696=1014.913,12.856,388.751,165.808,58.137,160.470
C06697=1014.920,13.105,388.738,165.811,58.128,160.469
C06698=1014.924,13.355,388.724,165.813,58.121,160.468
C06699=1014.929,13.605,388.711,165.815,58.112,160.467
C06700=1014.934,13.854,388.698,165.818,58.103,160.466
C06701=1014.939,14.104,388.685,165.819,58.094,160.465
C06702=1014.943,14.354,388.672,165.823,58.086,160.464
C06703=1014.949,14.603,388.658,165.825,58.077,160.463
C06704=1014.953,14.853,388.645,165.827,58.068,160.462
C06705=1014.959,15.102,388.631,165.829,58.059,160.461
C06706=1014.963,15.352,388.619,165.832,58.050,160.460
C06707=1014.969,15.601,388.605,165.833,58.042,160.458
C06708=1014.973,15.851,388.592,165.837,58.034,160.458
C06709=1014.979,16.100,388.578,165.839,58.025,160.456
C06710=1014.983,16.350,388.565,165.842,58.016,160.455
C06711=1014.989,16.600,388.552,165.843,58.007,160.454
C06712=1014.994,16.850,388.538,165.846,57.998,160.453
C06713=1014.999,17.099,388.526,165.849,57.989,160.452
C06714=1015.004,17.349,388.512,165.851,57.980,160.451
C06715=1015.009,17.598,388.499,165.853,57.972,160.450
C06716=1015.014,17.848,388.485,165.855,57.963,160.449
C06717=1015.019,18.097,388.472,165.858,57.954,160.448
C06718=1015.024,18.347,388.458,165.861,57.945,160.447
C06719=1015.029,18.596,388.446,165.862,57.937,160.445
C06720=1015.034,18.846,388.431,165.865,57.928,160.444
C06721=1015.039,19.096,388.417,165.868,57.920,160.444
C06722=1015.044,19.345,388.404,165.870,57.911,160.442
C06723=1015.049,19.595,388.391,165.872,57.902,160.441
C06724=1015.054,19.844,388.378,165.875,57.893,160.440
C06725=1015.058,20.094,388.363,165.878,57.884,160.439
C06726=1015.064,20.344,388.350,165.879,57.876,160.438
C06727=1015.068,20.593,388.337,165.882,57.867,160.437
C06728=1015.074,20.843,388.323,165.884,57.858,160.436
C06729=1015.079,21.092,388.309,165.887,57.849,160.435
C06730=1015.083,21.342,388.296,165.889,57.840,160.434
C06731=1015.089,21.592,388.282,165.891,57.832,160.433
C06732=1015.094,21.841,388.268,165.894,57.823,160.431
C06733=1015.099,22.091,388.255,165.897,57.814,160.430
C06734=1015.104,22.340,388.242,165.898,57.805,160.429
C06735=1015.108,22.590,388.227,165.901,57.796,160.428
C06736=1015.114,22.840,388.214,165.903,57.787,160.427
C06737=1015.118,23.089,388.201,165.906,57.778,160.426
C06738=1015.124,23.338,388.187,165.908,57.770,160.425
C06739=1015.129,23.589,388.173,165.910,57.761,160.424
C06740=1015.133,23.838,388.159,165.913,57.752,160.423
C06741=1015.139,24.087,388.146,165.916,57.743,160.422
C06742=1015.144,24.337,388.132,165.918,57.734,160.420
C06743=1015.149,24.586,388.119,165.919,57.725,160.419
C06744=1015.154,24.836,388.105,165.922,57.716,160.418
C06745=1015.159,25.086,388.091,165.925,57.707,160.417
C06746=1015.164,25.335,388.077,165.927,57.698,160.416
C06747=1015.169,25.585,388.064,165.930,57.689,160.415
C06748=1015.174,25.835,388.050,165.932,57.681,160.414
C06749=1015.180,26.115,388.034,165.935,57.671,160.413
C06750=1015.185,26.397,388.019,165.937,57.660,160.411
C06751=1015.191,26.677,388.003,165.939,57.650,160.410
C06752=1015.196,26.959,387.988,165.943,57.640,160.409
C06753=1015.202,27.208,387.974,165.945,57.632,160.408
C06754=1015.207,27.458,387.960,165.948,57.623,160.407
C06755=1015.212,27.708,387.945,165.950,57.614,160.405
C06756=1015.216,27.957,387.933,165.952,57.605,160.404
C06757=1015.221,28.207,387.918,165.955,57.596,160.403
C06758=1015.227,28.457,387.904,165.957,57.587,160.402
C06759=1015.231,28.707,387.890,165.959,57.578,160.401
C06760=1015.236,28.955,387.876,165.961,57.569,160.400
C06761=1015.241,29.205,387.862,165.964,57.561,160.399
C06762=1015.246,29.455,387.848,165.967,57.552,160.398
C06763=1015.251,29.704,387.835,165.970,57.543,160.397
C06764=1015.256,29.954,387.820,165.971,57.534,160.395
C06765=1015.262,30.203,387.806,165.973,57.525,160.394
C06766=1015.266,30.453,387.792,165.976,57.516,160.393
C06767=1015.271,30.702,387.778,165.979,57.507,160.392
C06768=1015.276,30.952,387.764,165.982,57.498,160.391
C06769=1015.281,31.201,387.750,165.983,57.490,160.390
C06770=1015.286,31.451,387.735,165.986,57.481,160.389
C06771=1015.292,31.701,387.722,165.988,57.471,160.387
C06772=1015.296,31.950,387.708,165.991,57.462,160.386
C06773=1015.301,32.200,387.694,165.993,57.453,160.385
C06774=1015.306,32.450,387.679,165.995,57.445,160.384
C06775=1015.311,32.699,387.665,165.997,57.435,160.383
C06776=1015.317,32.949,387.651,166.000,57.426,160.382
C06777=1015.321,33.198,387.637,166.003,57.418,160.381
C06778=1015.327,33.447,387.624,166.005,57.408,160.379
C06779=1015.331,33.697,387.609,166.008,57.399,160.378
C06780=1015.337,33.947,387.595,166.010,57.390,160.377
C06781=1015.342,34.196,387.580,166.012,57.382,160.376
C06782=1015.347,34.445,387.567,166.014,57.372,160.375
C06783=1015.351,34.695,387.552,166.017,57.363,160.374
C06784=1015.357,34.945,387.538,166.020,57.355,160.373
C06785=1015.362,35.194,387.524,166.022,57.345,160.371
C06786=1015.367,35.444,387.510,166.025,57.336,160.370
C06787=1015.372,35.694,387.495,166.027,57.327,160.369
C06788=1015.377,35.943,387.482,166.030,57.318,160.368
C06789=1015.381,36.193,387.467,166.032,57.309,160.367
C06790=1015.387,36.442,387.454,166.033,57.300,160.366
C06791=1015.392,36.691,387.438,166.036,57.291,160.364
C06792=1015.397,36.941,387.424,166.039,57.282,160.363
C06793=1015.402,37.191,387.410,166.042,57.273,160.362
C06794=1015.407,37.441,387.396,166.044,57.264,160.361
C06795=1015.411,37.689,387.381,166.046,57.255,160.360
C06796=1015.417,37.939,387.367,166.048,57.246,160.359
C06797=1015.422,38.189,387.353,166.051,57.237,160.358
C06798=1015.427,38.438,387.337,166.053,57.228,160.357
C06799=1015.431,38.688,387.323,166.056,57.219,160.356
C06800=1015.437,38.938,387.309,166.058,57.211,160.354
C06801=1015.442,39.187,387.295,166.060,57.201,160.353
C06802=1015.447,39.437,387.279,166.063,57.192,160.352
C06803=1015.452,39.686,387.266,166.066,57.183,160.351
C06804=1015.456,39.935,387.251,166.068,57.174,160.350
C06805=1015.461,40.185,387.236,166.071,57.165,160.349
C06806=1015.466,40.435,387.222,166.073,57.156,160.348
C06807=1015.471,40.684,387.208,166.075,57.147,160.346
C06808=1015.477,40.933,387.193,166.077,57.138,160.345
C06809=1015.484,41.306,387.171,166.081,57.124,160.343
C06810=1015.492,41.680,387.150,166.085,57.111,160.342
C06811=1015.499,42.053,387.127,166.088,57.097,160.340
C06812=1015.506,42.426,387.106,166.092,57.084,160.338
C06813=1015.512,42.741,387.087,166.095,57.072,160.337
C06814=1015.518,43.057,387.068,166.098,57.062,160.335
C06815=1015.523,43.307,387.053,166.101,57.053,160.334
C06816=1015.528,43.556,387.038,166.103,57.043,160.333
C06817=1015.533,43.806,387.024,166.106,57.034,160.332
C06818=1015.538,44.055,387.008,166.107,57.026,160.331
C06819=1015.543,44.304,386.993,166.110,57.017,160.330
C06820=1015.547,44.554,386.979,166.112,57.008,160.328
C06821=1015.553,44.803,386.964,166.115,56.999,160.327
C06822=1015.557,45.053,386.949,166.118,56.990,160.326
C06823=1015.562,45.303,386.934,166.119,56.981,160.325
C06824=1015.567,45.552,386.920,166.122,56.972,160.324
C06825=1015.572,45.802,386.904,166.125,56.963,160.323
C06826=1015.577,46.051,386.889,166.127,56.954,160.322
C06827=1015.582,46.301,386.875,166.130,56.945,160.321
C06828=1015.587,46.550,386.860,166.131,56.936,160.319
C06829=1015.592,46.799,386.844,166.134,56.927,160.318
C06830=1015.597,47.049,386.830,166.137,56.918,160.317
C06831=1015.602,47.299,386.815,166.139,56.909,160.316
C06832=1015.606,47.548,386.800,166.142,56.900,160.315
C06833=1015.612,47.798,386.785,166.144,56.891,160.314
C06834=1015.617,48.047,386.770,166.146,56.882,160.312
C06835=1015.621,48.297,386.755,166.149,56.873,160.311
C06836=1015.626,48.546,386.740,166.151,56.864,160.310
C06837=1015.631,48.795,386.725,166.154,56.855,160.309
C06838=1015.636,49.045,386.711,166.156,56.846,160.308
C06839=1015.641,49.295,386.695,166.159,56.837,160.307
C06840=1015.646,49.544,386.680,166.162,56.827,160.305
C06841=1015.651,49.794,386.666,166.163,56.819,160.304
C06842=1015.656,50.043,386.651,166.166,56.809,160.303
C06843=1015.661,50.292,386.636,166.168,56.801,160.302
C06844=1015.666,50.541,386.620,166.171,56.791,160.301
C06845=1015.671,50.791,386.606,166.174,56.782,160.300
C06846=1015.676,51.041,386.591,166.176,56.773,160.298
C06847=1015.681,51.290,386.576,166.179,56.764,160.297
C06848=1015.686,51.540,386.561,166.181,56.755,160.296
C06849=1015.691,51.789,386.546,166.184,56.746,160.295
C06850=1015.696,52.038,386.531,166.185,56.737,160.294
C06851=1015.701,52.288,386.515,166.188,56.727,160.292
C06852=1015.706,52.538,386.501,166.190,56.718,160.291
C06853=1015.711,52.787,386.486,166.193,56.709,160.290
C06854=1015.716,53.037,386.470,166.196,56.700,160.289
C06855=1015.721,53.286,386.455,166.198,56.691,160.288
C06856=1015.726,53.536,386.441,166.200,56.681,160.286
C06857=1015.731,53.785,386.426,166.203,56.672,160.285
C06858=1015.736,54.034,386.410,166.205,56.663,160.284
C06859=1015.740,54.284,386.395,166.208,56.653,160.283
C06860=1015.746,54.534,386.379,166.211,56.645,160.282
C06861=1015.751,54.784,386.365,166.213,56.635,160.281
C06862=1015.756,55.033,386.349,166.216,56.626,160.280
C06863=1015.761,55.282,386.334,166.218,56.617,160.278
C06864=1015.766,55.532,386.319,166.221,56.608,160.277
C06865=1015.771,55.781,386.304,166.223,56.598,160.276
C06866=1015.776,56.031,386.289,166.226,56.589,160.275
C06867=1015.781,56.280,386.274,166.228,56.580,160.273
C06868=1015.786,56.530,386.259,166.231,56.570,160.272
C06869=1015.791,56.779,386.244,166.233,56.562,160.271
C06870=1015.796,57.029,386.228,166.236,56.552,160.270
C06871=1015.802,57.278,386.213,166.238,56.543,160.269
C06872=1015.806,57.528,386.199,166.241,56.533,160.267
C06873=1015.811,57.777,386.184,166.243,56.524,160.266
C06874=1015.817,58.027,386.168,166.246,56.515,160.265
C06875=1015.822,58.307,386.151,166.248,56.505,160.263
C06876=1015.828,58.589,386.134,166.251,56.494,160.262
C06877=1015.834,58.870,386.117,166.253,56.484,160.261
C06878=1015.839,59.152,386.100,166.256,56.473,160.259
C06879=1015.845,59.401,386.085,166.259,56.464,160.258
C06880=1015.850,59.650,386.070,166.262,56.455,160.257
C06881=1015.855,59.900,386.054,166.264,56.445,160.256
C06882=1015.860,60.149,386.039,166.266,56.436,160.255
C06883=1015.865,60.399,386.024,166.269,56.426,160.253
C06884=1015.870,60.648,386.008,166.271,56.417,160.252
C06885=1015.875,60.897,385.993,166.273,56.408,160.251
C06886=1015.881,61.147,385.978,166.277,56.398,160.250
C06887=1015.886,61.396,385.963,166.280,56.389,160.249
C06888=1015.891,61.646,385.947,166.282,56.379,160.247
C06889=1015.896,61.895,385.932,166.285,56.370,160.246
C06890=1015.902,62.145,385.917,166.287,56.361,160.245
C06891=1015.907,62.394,385.901,166.289,56.351,160.244
C06892=1015.911,62.644,385.886,166.292,56.342,160.242
C06893=1015.916,62.893,385.871,166.295,56.333,160.241
C06894=1015.922,63.143,385.855,166.297,56.324,160.240
C06895=1015.926,63.393,385.839,166.300,56.314,160.239
C06896=1015.931,63.642,385.824,166.302,56.305,160.237
C06897=1015.937,63.892,385.809,166.305,56.296,160.237
C06898=1015.941,64.141,385.793,166.307,56.287,160.235
C06899=1015.946,64.391,385.778,166.310,56.277,160.234
C06900=1015.952,64.639,385.762,166.313,56.268,160.233
C06901=1015.956,64.890,385.746,166.315,56.259,160.232
C06902=1015.961,65.139,385.730,166.317,56.250,160.230
C06903=1015.966,65.388,385.715,166.319,56.241,160.229
C06904=1015.971,65.638,385.699,166.322,56.232,160.228
C06905=1015.977,65.887,385.683,166.324,56.222,160.227
C06906=1015.981,66.137,385.667,166.327,56.213,160.225
C06907=1015.986,66.386,385.652,166.329,56.204,160.224
C06908=1015.991,66.636,385.636,166.332,56.194,160.223
C06909=1015.996,66.885,385.621,166.335,56.186,160.222
C06910=1016.001,67.134,385.605,166.337,56.176,160.221
C06911=1016.006,67.384,385.589,166.340,56.167,160.219
C06912=1016.011,67.634,385.574,166.342,56.157,160.218
C06913=1016.016,67.883,385.558,166.345,56.149,160.217
C06914=1016.022,68.133,385.542,166.348,56.139,160.216
C06915=1016.026,68.382,385.526,166.350,56.130,160.215
C06916=1016.031,68.631,385.511,166.352,56.120,160.213
C06917=1016.036,68.880,385.494,166.355,56.112,160.212
C06918=1016.041,69.130,385.479,166.358,56.102,160.211
C06919=1016.046,69.379,385.462,166.360,56.093,160.210
C06920=1016.051,69.629,385.447,166.363,56.083,160.209
C06921=1016.056,69.879,385.431,166.366,56.075,160.208
C06922=1016.060,70.128,385.414,166.368,56.065,160.206
C06923=1016.066,70.378,385.399,166.371,56.056,160.205
C06924=1016.070,70.627,385.383,166.373,56.047,160.204
C06925=1016.076,70.876,385.367,166.376,56.037,160.203
C06926=1016.081,71.126,385.351,166.378,56.029,160.202
C06927=1016.086,71.375,385.335,166.380,56.020,160.200
C06928=1016.090,71.624,385.319,166.383,56.010,160.199
C06929=1016.095,71.874,385.303,166.385,56.001,160.198
C06930=1016.101,72.123,385.287,166.388,55.991,160.197
C06931=1016.105,72.372,385.271,166.391,55.983,160.196
C06932=1016.111,72.622,385.255,166.393,55.973,160.194
C06933=1016.115,72.872,385.240,166.396,55.964,160.193
C06934=1016.120,73.122,385.223,166.398,55.955,160.192
C06935=1016.125,73.371,385.208,166.401,55.945,160.191
C06936=1016.130,73.620,385.191,166.403,55.936,160.189
C06937=1016.136,73.870,385.176,166.406,55.927,160.188
C06938=1016.140,74.119,385.159,166.409,55.918,160.187
C06939=1016.146,74.400,385.141,166.412,55.907,160.186
C06940=1016.152,74.682,385.123,166.415,55.897,160.184
C06941=1016.158,74.962,385.104,166.418,55.886,160.183
C06942=1016.163,75.244,385.086,166.421,55.876,160.182
C06943=1016.168,75.493,385.071,166.423,55.866,160.180
C06944=1016.173,75.743,385.054,166.426,55.857,160.179
C06945=1016.177,75.992,385.038,166.428,55.848,160.178
C06946=1016.183,76.242,385.022,166.431,55.838,160.177
C06947=1016.188,76.491,385.006,166.433,55.829,160.175
C06948=1016.192,76.740,384.990,166.436,55.820,160.174
C06949=1016.198,76.990,384.974,166.439,55.811,160.173
C06950=1016.203,77.239,384.957,166.442,55.802,160.172
C06951=1016.208,77.489,384.941,166.444,55.792,160.171
C06952=1016.212,77.738,384.925,166.447,55.783,160.169
C06953=1016.217,77.987,384.908,166.449,55.775,160.168
C06954=1016.222,78.237,384.892,166.451,55.765,160.167
C06955=1016.227,78.487,384.875,166.454,55.756,160.166
C06956=1016.232,78.736,384.859,166.456,55.747,160.165
C06957=1016.237,78.985,384.842,166.459,55.737,160.163
C06958=1016.242,79.235,384.827,166.462,55.729,160.162
C06959=1016.247,79.484,384.810,166.464,55.719,160.161
C06960=1016.252,79.733,384.793,166.467,55.710,160.160
C06961=1016.256,79.982,384.777,166.470,55.701,160.159
C06962=1016.261,80.232,384.761,166.472,55.691,160.157
C06963=1016.266,80.481,384.744,166.475,55.683,160.156
C06964=1016.271,80.731,384.727,166.478,55.673,160.155
C06965=1016.276,80.980,384.711,166.480,55.664,160.154
C06966=1016.281,81.230,384.694,166.483,55.655,160.153
C06967=1016.286,81.479,384.679,166.485,55.645,160.152
C06968=1016.291,81.729,384.662,166.488,55.636,160.150
C06969=1016.296,81.978,384.645,166.491,55.627,160.149
C06970=1016.301,82.227,384.629,166.494,55.618,160.148
C06971=1016.306,82.477,384.612,166.496,55.609,160.147
C06972=1016.310,82.726,384.596,166.499,55.599,160.146
C06973=1016.316,82.976,384.579,166.501,55.590,160.144
C06974=1016.320,83.225,384.563,166.504,55.581,160.143
C06975=1016.325,83.475,384.546,166.507,55.571,160.142
C06976=1016.330,83.724,384.529,166.509,55.562,160.141
C06977=1016.336,83.973,384.513,166.512,55.553,160.139
C06978=1016.341,84.222,384.497,166.514,55.543,160.138
C06979=1016.345,84.472,384.480,166.517,55.534,160.137
C06980=1016.350,84.721,384.464,166.520,55.525,160.136
C06981=1016.355,84.971,384.447,166.522,55.516,160.135
C06982=1016.361,85.221,384.430,166.525,55.506,160.133
C06983=1016.365,85.470,384.414,166.527,55.497,160.132
C06984=1016.370,85.719,384.397,166.531,55.488,160.131
C06985=1016.375,85.968,384.380,166.533,55.479,160.130
C06986=1016.380,86.218,384.364,166.536,55.470,160.129
C06987=1016.385,86.467,384.347,166.538,55.460,160.127
C06988=1016.390,86.717,384.332,166.541,55.451,160.126
C06989=1016.396,86.966,384.315,166.544,55.442,160.125
C06990=1016.400,87.215,384.298,166.546,55.432,160.124
C06991=1016.405,87.465,384.281,166.549,55.423,160.123
C06992=1016.410,87.714,384.265,166.551,55.414,160.121
C06993=1016.415,87.964,384.248,166.554,55.404,160.120
C06994=1016.421,88.213,384.231,166.556,55.395,160.119
C06995=1016.425,88.462,384.215,166.560,55.385,160.117
C06996=1016.430,88.712,384.198,166.562,55.376,160.116
C06997=1016.436,88.962,384.181,166.565,55.366,160.115
C06998=1016.440,89.211,384.165,166.568,55.358,160.114
C06999=1016.445,89.460,384.148,166.571,55.348,160.113
C07000=1016.450,89.710,384.130,166.572,55.340,160.111
C07001=1016.454,89.959,384.114,166.575,55.330,160.110
C07002=1016.460,90.208,384.096,166.578,55.321,160.109
C07003=1016.465,90.490,384.078,166.581,55.311,160.108
C07004=1016.471,90.771,384.059,166.584,55.300,160.106
C07005=1016.476,91.052,384.040,166.587,55.290,160.105
C07006=1016.482,91.333,384.020,166.590,55.279,160.104
C07007=1016.487,91.583,384.003,166.593,55.270,160.103
C07008=1016.491,91.832,383.986,166.596,55.261,160.101
C07009=1016.497,92.081,383.969,166.598,55.252,160.100
C07010=1016.502,92.331,383.952,166.601,55.242,160.099
C07011=1016.506,92.580,383.935,166.604,55.233,160.098
C07012=1016.511,92.830,383.918,166.607,55.224,160.097
C07013=1016.516,93.080,383.901,166.610,55.215,160.095
C07014=1016.521,93.328,383.884,166.612,55.206,160.094
C07015=1016.526,93.578,383.867,166.615,55.197,160.093
C07016=1016.531,93.828,383.850,166.618,55.187,160.092
C07017=1016.535,94.077,383.833,166.620,55.178,160.091
C07018=1016.541,94.326,383.816,166.623,55.169,160.089
C07019=1016.546,94.575,383.799,166.626,55.160,160.088
C07020=1016.550,94.825,383.782,166.628,55.150,160.087
C07021=1016.555,95.074,383.765,166.631,55.141,160.086
C07022=1016.561,95.323,383.747,166.634,55.132,160.085
C07023=1016.566,95.573,383.730,166.636,55.123,160.083
C07024=1016.570,95.822,383.713,166.639,55.113,160.082
C07025=1016.575,96.072,383.697,166.642,55.104,160.081
C07026=1016.581,96.321,383.679,166.644,55.095,160.080
C07027=1016.586,96.571,383.662,166.647,55.086,160.078
C07028=1016.590,96.820,383.645,166.650,55.076,160.077
C07029=1016.595,97.069,383.627,166.653,55.067,160.076
C07030=1016.600,97.318,383.611,166.655,55.058,160.075
C07031=1016.605,97.567,383.594,166.659,55.048,160.074
C07032=1016.611,97.816,383.577,166.662,55.039,160.073
C07033=1016.615,98.066,383.559,166.664,55.030,160.071
C07034=1016.620,98.316,383.542,166.667,55.021,160.070
C07035=1016.626,98.565,383.525,166.669,55.011,160.069
C07036=1016.630,98.814,383.508,166.672,55.001,160.067
C07037=1016.635,99.064,383.491,166.675,54.992,160.066
C07038=1016.640,99.313,383.473,166.678,54.984,160.065
C07039=1016.645,99.563,383.456,166.681,54.974,160.064
C07040=1016.650,99.811,383.439,166.683,54.965,160.063
C07041=1016.654,100.061,383.421,166.686,54.956,160.062
C07042=1016.660,100.310,383.404,166.689,54.947,160.060
C07043=1016.664,100.560,383.386,166.692,54.937,160.059
C07044=1016.670,100.809,383.369,166.694,54.928,160.058
C07045=1016.674,101.059,383.351,166.697,54.919,160.057
C07046=1016.679,101.308,383.334,166.700,54.910,160.056
C07047=1016.684,101.557,383.316,166.703,54.901,160.054
C07048=1016.688,101.807,383.298,166.705,54.891,160.053
C07049=1016.694,102.056,383.281,166.708,54.882,160.052
C07050=1016.698,102.305,383.264,166.711,54.873,160.051
C07051=1016.703,102.554,383.246,166.714,54.864,160.050
C07052=1016.708,102.804,383.229,166.717,54.855,160.049
C07053=1016.713,103.053,383.211,166.720,54.846,160.047
C07054=1016.718,103.303,383.193,166.722,54.837,160.046
C07055=1016.723,103.552,383.176,166.725,54.828,160.045
C07056=1016.728,103.801,383.158,166.728,54.818,160.044
C07057=1016.733,104.051,383.141,166.731,54.809,160.043
C07058=1016.737,104.300,383.123,166.733,54.800,160.041
C07059=1016.743,104.549,383.106,166.736,54.791,160.040
C07060=1016.747,104.799,383.088,166.739,54.782,160.039
C07061=1016.752,105.048,383.070,166.742,54.772,160.038
C07062=1016.757,105.297,383.053,166.744,54.763,160.037
C07063=1016.762,105.547,383.035,166.747,54.754,160.035
C07064=1016.767,105.796,383.018,166.750,54.745,160.034
C07065=1016.772,106.045,383.000,166.753,54.736,160.033
C07066=1016.777,106.295,382.983,166.757,54.726,160.032
C07067=1016.782,106.577,382.963,166.758,54.715,160.030
C07068=1016.789,106.858,382.943,166.762,54.705,160.029
C07069=1016.794,107.139,382.923,166.765,54.695,160.028
C07070=1016.799,107.421,382.903,166.768,54.685,160.026
C07071=1016.804,107.670,382.885,166.772,54.675,160.025
C07072=1016.809,107.920,382.867,166.775,54.666,160.024
C07073=1016.815,108.169,382.850,166.777,54.656,160.023
C07074=1016.819,108.419,382.832,166.780,54.647,160.021
C07075=1016.824,108.667,382.815,166.783,54.638,160.020
C07076=1016.829,108.916,382.797,166.786,54.628,160.019
C07077=1016.834,109.166,382.780,166.788,54.619,160.018
C07078=1016.839,109.415,382.762,166.791,54.610,160.017
C07079=1016.844,109.665,382.744,166.794,54.601,160.015
C07080=1016.849,109.914,382.726,166.797,54.592,160.014
C07081=1016.854,110.163,382.708,166.800,54.583,160.013
C07082=1016.859,110.412,382.690,166.802,54.573,160.012
C07083=1016.863,110.662,382.672,166.805,54.564,160.011
C07084=1016.869,110.911,382.655,166.809,54.555,160.010
C07085=1016.874,111.161,382.637,166.812,54.546,160.008
C07086=1016.878,111.410,382.619,166.815,54.536,160.007
C07087=1016.883,111.659,382.600,166.818,54.527,160.006
C07088=1016.889,111.909,382.583,166.820,54.518,160.005
C07089=1016.893,112.158,382.565,166.823,54.509,160.004
C07090=1016.898,112.407,382.546,166.826,54.500,160.002
C07091=1016.903,112.657,382.528,166.829,54.491,160.001
C07092=1016.908,112.906,382.510,166.832,54.482,160.000
C07093=1016.912,113.155,382.492,166.835,54.473,159.999
C07094=1016.917,113.404,382.474,166.838,54.464,159.998
C07095=1016.922,113.653,382.456,166.841,54.455,159.997
C07096=1016.926,113.903,382.438,166.844,54.446,159.996
C07097=1016.931,114.152,382.420,166.846,54.436,159.994
C07098=1016.936,114.401,382.402,166.849,54.427,159.993
C07099=1016.941,114.651,382.383,166.852,54.418,159.992
C07100=1016.945,114.900,382.365,166.855,54.410,159.991
C07101=1016.951,115.149,382.346,166.858,54.401,159.990
C07102=1016.955,115.398,382.328,166.861,54.391,159.989
C07103=1016.959,115.648,382.309,166.864,54.382,159.987
C07104=1016.964,115.897,382.291,166.867,54.373,159.986
C07105=1016.969,116.146,382.273,166.870,54.364,159.985
C07106=1016.974,116.396,382.255,166.873,54.355,159.984
C07107=1016.978,116.645,382.237,166.875,54.346,159.983
C07108=1016.983,116.895,382.219,166.878,54.337,159.982
C07109=1016.988,117.143,382.200,166.881,54.328,159.980
C07110=1016.993,117.393,382.182,166.884,54.318,159.979
C07111=1016.998,117.642,382.163,166.887,54.309,159.978
C07112=1017.003,117.891,382.145,166.890,54.301,159.977
C07113=1017.008,118.141,382.127,166.893,54.292,159.976
C07114=1017.013,118.390,382.108,166.896,54.283,159.975
C07115=1017.018,118.639,382.090,166.899,54.274,159.973
C07116=1017.023,118.889,382.072,166.902,54.264,159.972
C07117=1017.027,119.138,382.053,166.905,54.255,159.971
C07118=1017.032,119.387,382.035,166.908,54.246,159.970
C07119=1017.037,119.636,382.016,166.910,54.237,159.969
C07120=1017.042,119.886,381.998,166.913,54.228,159.968
C07121=1017.047,120.135,381.980,166.916,54.219,159.966
C07122=1017.052,120.384,381.962,166.919,54.210,159.965
C07123=1017.056,120.634,381.944,166.923,54.200,159.964
C07124=1017.062,120.882,381.925,166.926,54.191,159.963
C07125=1017.066,121.132,381.907,166.929,54.182,159.962
C07126=1017.071,121.381,381.888,166.932,54.173,159.961
C07127=1017.077,121.630,381.869,166.935,54.164,159.959
C07128=1017.082,121.880,381.851,166.938,54.155,159.958
C07129=1017.086,122.129,381.833,166.940,54.146,159.957
C07130=1017.091,122.379,381.815,166.943,54.137,159.956
C07131=1017.096,122.660,381.794,166.947,54.126,159.955
C07132=1017.102,122.942,381.773,166.950,54.115,159.953
C07133=1017.107,123.223,381.752,166.953,54.105,159.952
C07134=1017.113,123.504,381.731,166.957,54.095,159.951
C07135=1017.118,123.754,381.713,166.960,54.086,159.949
C07136=1017.123,124.003,381.694,166.964,54.077,159.948
C07137=1017.128,124.253,381.676,166.967,54.067,159.947
C07138=1017.133,124.502,381.658,166.969,54.058,159.946
C07139=1017.138,124.751,381.639,166.972,54.049,159.945
C07140=1017.143,125.000,381.621,166.975,54.040,159.944
C07141=1017.149,125.249,381.601,166.978,54.030,159.942
C07142=1017.153,125.499,381.583,166.981,54.021,159.941
C07143=1017.157,125.748,381.564,166.985,54.012,159.940
C07144=1017.162,125.997,381.545,166.988,54.003,159.939
C07145=1017.167,126.246,381.527,166.991,53.994,159.938
C07146=1017.172,126.496,381.509,166.993,53.985,159.936
C07147=1017.178,126.745,381.490,166.996,53.976,159.935
C07148=1017.182,126.995,381.472,166.999,53.967,159.934
C07149=1017.188,127.243,381.453,167.003,53.957,159.933
C07150=1017.192,127.493,381.435,167.006,53.948,159.932
C07151=1017.197,127.742,381.417,167.009,53.939,159.931
C07152=1017.203,127.991,381.397,167.012,53.929,159.929
C07153=1017.208,128.241,381.379,167.015,53.920,159.928
C07154=1017.213,128.490,381.360,167.019,53.911,159.927
C07155=1017.217,128.739,381.342,167.022,53.902,159.926
C07156=1017.223,128.988,381.323,167.025,53.893,159.925
C07157=1017.228,129.238,381.305,167.028,53.884,159.924
C07158=1017.233,129.486,381.286,167.031,53.875,159.922
C07159=1017.237,129.736,381.267,167.035,53.865,159.921
C07160=1017.243,129.986,381.248,167.038,53.856,159.920
C07161=1017.248,130.235,381.230,167.040,53.847,159.919
C07162=1017.252,130.484,381.210,167.043,53.838,159.918
C07163=1017.258,130.733,381.191,167.046,53.829,159.917
C07164=1017.262,130.983,381.172,167.049,53.820,159.915
C07165=1017.267,131.232,381.153,167.052,53.811,159.914
C07166=1017.272,131.480,381.134,167.055,53.802,159.913
C07167=1017.276,131.731,381.115,167.058,53.793,159.912
C07168=1017.282,131.980,381.096,167.061,53.784,159.911
C07169=1017.286,132.229,381.077,167.065,53.774,159.910
C07170=1017.291,132.478,381.059,167.068,53.765,159.909
C07171=1017.296,132.728,381.039,167.071,53.756,159.907
C07172=1017.301,132.976,381.020,167.074,53.747,159.906
C07173=1017.306,133.225,381.001,167.077,53.738,159.905
C07174=1017.310,133.476,380.982,167.081,53.730,159.904
C07175=1017.315,133.724,380.963,167.084,53.721,159.903
C07176=1017.320,133.973,380.944,167.087,53.712,159.902
C07177=1017.325,134.222,380.925,167.091,53.702,159.901
C07178=1017.330,134.472,380.906,167.094,53.693,159.900
C07179=1017.335,134.721,380.887,167.097,53.684,159.898
C07180=1017.340,134.970,380.868,167.100,53.675,159.897
C07181=1017.345,135.220,380.848,167.103,53.666,159.896
C07182=1017.350,135.468,380.829,167.106,53.657,159.895
C07183=1017.354,135.718,380.811,167.110,53.648,159.894
C07184=1017.360,135.967,380.791,167.113,53.639,159.893
C07185=1017.364,136.216,380.772,167.116,53.630,159.892
C07186=1017.369,136.465,380.753,167.119,53.621,159.890
C07187=1017.375,136.715,380.734,167.122,53.612,159.889
C07188=1017.379,136.964,380.714,167.125,53.603,159.888
C07189=1017.385,137.213,380.695,167.128,53.594,159.887
C07190=1017.389,137.463,380.676,167.132,53.585,159.886
C07191=1017.394,137.712,380.657,167.135,53.576,159.885
C07192=1017.399,137.961,380.637,167.138,53.567,159.884
C07193=1017.403,138.210,380.618,167.141,53.558,159.882
C07194=1017.408,138.459,380.599,167.144,53.549,159.881
C07195=1017.414,138.741,380.577,167.148,53.538,159.880
C07196=1017.419,139.022,380.555,167.151,53.528,159.879
C07197=1017.424,139.304,380.533,167.155,53.518,159.877
C07198=1017.430,139.585,380.511,167.159,53.508,159.876
C07199=1017.434,139.834,380.492,167.162,53.499,159.875
C07200=1017.440,140.084,380.472,167.166,53.490,159.874
C07201=1017.444,140.333,380.453,167.169,53.481,159.873
C07202=1017.449,140.583,380.433,167.172,53.472,159.872
C07203=1017.454,140.831,380.414,167.175,53.464,159.871
C07204=1017.459,141.080,380.394,167.179,53.455,159.870
C07205=1017.464,141.329,380.374,167.182,53.446,159.868
C07206=1017.469,141.578,380.355,167.186,53.436,159.867
C07207=1017.474,141.828,380.335,167.189,53.427,159.866
C07208=1017.478,142.077,380.316,167.192,53.418,159.865
C07209=1017.484,142.326,380.297,167.195,53.409,159.864
C07210=1017.488,142.575,380.277,167.198,53.400,159.863
C07211=1017.493,142.825,380.257,167.201,53.391,159.862
C07212=1017.498,143.074,380.238,167.205,53.382,159.861
C07213=1017.503,143.323,380.219,167.208,53.373,159.859
C07214=1017.508,143.572,380.198,167.211,53.364,159.858
C07215=1017.512,143.821,380.179,167.214,53.355,159.857
C07216=1017.518,144.071,380.160,167.217,53.346,159.856
C07217=1017.522,144.320,380.140,167.222,53.337,159.855
C07218=1017.527,144.569,380.120,167.225,53.329,159.854
C07219=1017.532,144.818,380.102,167.228,53.320,159.853
C07220=1017.538,145.067,380.081,167.231,53.311,159.852
C07221=1017.542,145.316,380.061,167.234,53.302,159.850
C07222=1017.548,145.566,380.042,167.238,53.293,159.849
C07223=1017.552,145.815,380.023,167.242,53.284,159.848
C07224=1017.557,146.064,380.002,167.245,53.275,159.847
C07225=1017.562,146.313,379.983,167.248,53.266,159.846
C07226=1017.567,146.563,379.963,167.251,53.257,159.845
C07227=1017.571,146.812,379.943,167.255,53.247,159.844
C07228=1017.576,147.061,379.923,167.259,53.239,159.843
C07229=1017.581,147.310,379.903,167.262,53.230,159.842
C07230=1017.586,147.559,379.884,167.265,53.221,159.841
C07231=1017.592,147.808,379.864,167.268,53.212,159.839
C07232=1017.596,148.057,379.844,167.271,53.203,159.838
C07233=1017.601,148.307,379.824,167.275,53.194,159.837
C07234=1017.605,148.556,379.804,167.278,53.185,159.836
C07235=1017.610,148.805,379.784,167.282,53.177,159.835
C07236=1017.615,149.054,379.764,167.285,53.168,159.834
C07237=1017.620,149.304,379.744,167.288,53.159,159.833
C07238=1017.625,149.552,379.724,167.292,53.150,159.832
C07239=1017.630,149.802,379.704,167.295,53.141,159.831
C07240=1017.635,150.051,379.684,167.298,53.132,159.829
C07241=1017.639,150.300,379.664,167.302,53.123,159.828
C07242=1017.644,150.549,379.644,167.305,53.115,159.827
C07243=1017.649,150.798,379.624,167.309,53.105,159.826
C07244=1017.654,151.048,379.604,167.312,53.097,159.825
C07245=1017.658,151.296,379.584,167.316,53.088,159.824
C07246=1017.663,151.546,379.564,167.319,53.079,159.823
C07247=1017.669,151.795,379.544,167.323,53.069,159.822
C07248=1017.673,152.044,379.524,167.326,53.061,159.821
C07249=1017.678,152.293,379.504,167.330,53.052,159.820
C07250=1017.684,152.542,379.484,167.333,53.043,159.819
C07251=1017.689,152.791,379.464,167.336,53.035,159.818
C07252=1017.693,153.041,379.443,167.340,53.025,159.816
C07253=1017.697,153.290,379.424,167.343,53.016,159.815
C07254=1017.703,153.539,379.403,167.346,53.007,159.814
C07255=1017.708,153.788,379.383,167.350,52.999,159.813
C07256=1017.712,154.037,379.363,167.354,52.990,159.812
C07257=1017.718,154.286,379.343,167.357,52.981,159.811
C07258=1017.723,154.536,379.323,167.360,52.972,159.810
C07259=1017.728,154.817,379.299,167.364,52.962,159.809
C07260=1017.733,155.099,379.277,167.368,52.952,159.807
C07261=1017.739,155.380,379.254,167.372,52.942,159.806
C07262=1017.744,155.662,379.231,167.376,52.932,159.805
C07263=1017.749,155.910,379.211,167.380,52.924,159.804
C07264=1017.754,156.159,379.190,167.383,52.915,159.803
C07265=1017.759,156.408,379.170,167.386,52.906,159.802
C07266=1017.764,156.657,379.150,167.391,52.897,159.801
C07267=1017.769,156.906,379.130,167.394,52.888,159.800
C07268=1017.774,157.156,379.108,167.397,52.880,159.799
C07269=1017.778,157.405,379.089,167.401,52.871,159.798
C07270=1017.783,157.654,379.068,167.405,52.862,159.797
C07271=1017.788,157.903,379.048,167.408,52.853,159.795
C07272=1017.794,158.152,379.027,167.411,52.844,159.794
C07273=1017.798,158.401,379.008,167.415,52.835,159.793
C07274=1017.803,158.650,378.987,167.419,52.826,159.792
C07275=1017.808,158.900,378.966,167.422,52.818,159.791
C07276=1017.812,159.149,378.945,167.425,52.809,159.790
C07277=1017.817,159.398,378.925,167.429,52.801,159.789
C07278=1017.821,159.647,378.904,167.432,52.792,159.788
C07279=1017.827,159.896,378.883,167.437,52.783,159.787
C07280=1017.831,160.145,378.862,167.440,52.774,159.786
C07281=1017.835,160.394,378.841,167.444,52.766,159.785
C07282=1017.841,160.643,378.820,167.447,52.757,159.784
C07283=1017.845,160.892,378.799,167.450,52.748,159.783
C07284=1017.850,161.141,378.779,167.454,52.740,159.782
C07285=1017.854,161.390,378.757,167.458,52.731,159.781
C07286=1017.859,161.640,378.736,167.462,52.723,159.780
C07287=1017.864,161.889,378.716,167.465,52.714,159.779
C07288=1017.868,162.137,378.695,167.468,52.705,159.778
